// TIA Portal project "Trabajo_plantilla" (V14)
// Plantilla para la realización de la parte de programación de la asignatura de Automatización

(* hardware
DEVICE "S71500/ET200MP station_16"  S7-1500 station
   slot 0: "Perfil soporte_0"  Rack  6ES7 590-1***0-0AA0
   slot 1: "AUTO_CELDA_DE_CORTE"  CPU 1516F-3 PN/DP  6ES7 516-3FN00-0AB0  V1.8
      slot 3: "Display de la CPU_1"  6ES7591-1BA00-0AA0
   slot 2: "DI 32x24VDC BA_1"  DI 32x24VDC BA  6ES7 521-1BL10-0AA0  V1.0
   slot 3: "DQ 32x24VDC/0.5A BA_1"  DQ 32x24VDC/0.5A BA  6ES7 522-1BL10-0AA0  V1.0
   slot 4: "DI 32x24VDC BA_2"  DI 32x24VDC BA  6ES7 521-1BL10-0AA0  V1.0
*)

// ===== PLC "AUTO_CELDA_DE_CORTE"  CPU 1516F-3 PN/DP =====

VAR_GLOBAL   // PLC tag table "Tests Unitarios"
   "Tag_1" AT %M20.0 : Bool;
   "Tag_2" AT %M20.1 : Bool;
   "Tag_3" AT %M20.2 : Bool;
   "Tag_4" AT %M20.3 : Bool;
   "Tag_6" AT %M20.5 : Bool;
   "Tag_7" AT %M20.6 : Bool;
   "Tag_5" AT %M20.4 : Bool;
   "Tag_8" AT %M20.7 : Bool;
   "Tag_9" AT %M21.0 : Bool;
   "Tag_10" AT %M21.1 : Bool;
   "Tag_12" AT %MD22 : Real;
   "Tag_11" AT %M21.2 : Bool;
   "Tag_13" AT %M21.3 : Bool;
   "Tag_14" AT %M21.4 : Bool;
   "Tag_15" AT %M21.5 : Bool;
   "Tag_16" AT %M21.6 : Bool;
   "Tag_17" AT %M21.7 : Bool;
END_VAR

VAR_GLOBAL   // PLC tag table "Entradas"
   "SB2_inferior" AT %E3.5 : Bool;   // Sensor de presencia que detecta la legada de piezas al brazo 2 (derecha) desde la cinta inferior
   "SB2_superior" AT %E3.4 : Bool;   // Sensor de presencia que detecta la legada de piezas al brazo 2 (derecha) desde la cinta superior
   "SB1_inferior" AT %E3.3 : Bool;   // Sensor de presencia que detecta la legada de piezas al brazo 1 (izquierda) desde la cinta inferior
   "SB1_superior" AT %E3.2 : Bool;   // Sensor de presencia que detecta la legada de piezas al brazo 1 (izquierda) desde la cinta superior
   "pieza_válida_serigrafía" AT %E2.7 : Bool;   // Aviso del lector de códigos correspondiente de que la pieza detectada debe ser incorporada a la máquina de serigrafía
   "pieza_válida_laminado" AT %E4.1 : Bool;   // Aviso del lector de códigos correspondiente de que la pieza detectada debe ser incorporada a la máquina de laminado
   "pieza_válida_corte" AT %E4.0 : Bool;   // Aviso del lector de códigos correspondiente de que la pieza detectada debe ser incorporada a la máquina de corte
   "FC3_E" AT %E0.7 : Bool;   // Fin de carrera del pistón de alimentación de la máquina de serigrafía (expandido)
   "FC3_C" AT %E0.6 : Bool;   // Fin de carrera del pistón de alimentación de la máquina de serigrafía (comprimido)
   "FC2_E" AT %E0.5 : Bool;   // Fin de carrera del pistón de alimentación de la máquina de laminado (expandido)
   "FC2_C" AT %E0.4 : Bool;   // Fin de carrera del pistón de alimentación de la máquina de laminado (comprimido)
   "FC1_E" AT %E0.3 : Bool;   // Fin de carrera del pistón de alimentación de la máquina de corte (expandido)
   "FC1_C" AT %E0.2 : Bool;   // Fin de carrera del pistón de alimentación de la máquina de corte (comprimido)
   "SS0" AT %E4.2 : Bool;   // Sensor de presencia de la cinta de alimentación, sobre la máquina de serigrafiado
   "SL0" AT %E3.7 : Bool;   // Sensor de presencia de la cinta de alimentación, sobre la máquina de laminado
   "SC0" AT %E3.6 : Bool;   // Sensor de presencia de la cinta de alimentación, sobre la máquina de corte
   "SS3_Derecha" AT %E2.4 : Bool;   // Sensor de incorporación a la cinta de evacuación de la serigrafiadora (derecha)
   "SL3_Derecha" AT %E3.1 : Bool;   // Sensor de incorporación a la cinta de evacuación de la laminadora (derecha)
   "SC3_Derecha" AT %E3.0 : Bool;   // Sensor de incorporación a la cinta de evacuación de la máquina de corte (a la derecha)
   "MB" AT %E2.6 : Bool;   // Señal de Activación del Modo de Marcha B
   "MA" AT %E2.5 : Bool;   // Señal de Activación del Modo de Marcha A
   "OFF" AT %E0.1 : Bool;   // Señal de parada controlada
   "SS3_Izquierda" AT %E2.3 : Bool;   // Sensor de incorporación a la cinta de evacuación de la serigrafiadora (izquierda)
   "SS2" AT %E2.2 : Bool;   // Sensor a la salida de la serigrafiadora
   "SS1" AT %E2.1 : Bool;   // Sensor de presencia a la entrada de la serigrafiadora
   "SL3_Izquierda" AT %E2.0 : Bool;   // Sensor de incorporación a la cinta de evacuación de la laminadora (izquierda)
   "SL2" AT %E1.7 : Bool;   // Sensor a la salida de la laminadora
   "SL1" AT %E1.6 : Bool;   // Sensor de presencia a la entrada de la laminadora
   "SC3_Izquierda" AT %E1.5 : Bool;   // Sensor de incorporación a la cinta de evacuación de la máquina de corte (a la izquierda)
   "SC2" AT %E1.4 : Bool;   // Sensor a la salida de la máquina de corte
   "SC1" AT %E1.3 : Bool;   // Sensor de presencia a la entrada de la máquina de corte
   "ON" AT %E0.0 : Bool;   // Puesta en marcha del sistema
   "señal_pirómetro" AT %EW6 : Int;   // Señal analógica del sensor de temperatura
   "Rearme" AT %E1.0 : Bool;   // Señal de activación del rearme
   "EMER" AT %E1.1 : Bool;   // Señal de activación del estado de emergencia
END_VAR

VAR_GLOBAL   // PLC tag table "Actuadores"
   "EXTRAER_INFERIOR_B2" AT %A0.2 : Bool;   // Actuador que engloba la operación de extracción de piezas por la cinta inferior del brazo 2
   "EXTRAER_SUPERIOR_B2" AT %A0.1 : Bool;   // Actuador que engloba la operación de extracción de piezas por la cinta superior del brazo 2
   "ALIMENTAR_B2" AT %A0.0 : Bool;   // Actuador que engloba la operación de alimentación del brazo 2
   "EXTRAER_INFERIOR_B1" AT %A0.5 : Bool;   // Actuador que engloba la operación de extracción de piezas por la cinta inferior del brazo 1
   "EXTRAER_SUPERIOR_B1" AT %A0.4 : Bool;   // Actuador que engloba la operación de extracción de piezas por la cinta superior del brazo 1
   "ALIMENTAR_B1" AT %A0.3 : Bool;   // Actuador que engloba la operación de alimentación del brazo 1
   "CINTA_VOLCADO_Corte" AT %A2.2 : Bool;   // Actuador que activa la cinta de volcado de piezas de la máquina de corte
   "COMP3" AT %A1.3 : Bool;   // Actuador que efectúa la compresión del cilindro de alimentación de la máquina de serigrafía
   "EXP3" AT %A1.2 : Bool;   // Actuador que efectúa la expansión del cilindro de alimentación de la máquina de serigrafía
   "COMP2" AT %A1.1 : Bool;   // Actuador que efectúa la compresión del cilindro de alimentación de la máquina de laminado
   "EXP2" AT %A1.0 : Bool;   // Actuador que efectúa la expansión del cilindro de alimentación de la máquina de laminado
   "COMP1" AT %A0.7 : Bool;   // Actuador que efectúa la compresión del cilindro de alimentación de la máquina de corte
   "EXP1" AT %A0.6 : Bool;   // Actuador que efectúa la expansión del cilindro de alimentación de la máquina de corte
   "MÁQUINA_SERIGRAFIADO_ON" AT %A2.4 : Bool;   // Actuador que engloba el funcionamiento de la CNC de serigrafía
   "MÁQUINA_LAMINADO_ON" AT %A2.5 : Bool;   // Actuador que engloba el funcionamiento de la CNC de laminado
   "MÁQUINA_CORTE_ON" AT %A2.6 : Bool;   // Actuador que engloba el funcionamiento de la CNC de corte
   "CINTA_VOLCADO_Laminado" AT %A2.3 : Bool;   // Actuador que activa la cinta de volcado de piezas de la máquina de laminado
   "LÁMPARA_IR" AT %A2.0 : Bool;   // Lámpara infrarroja para el precalentado de piezas en la laminadora
   "CINTA_VOLCADO_Serigrafiado" AT %A2.1 : Bool;   // Actuador que activa la cinta de volcado de piezas de la máquina de serigrafiado
   "CINTA1_H" AT %A1.4 : Bool;   // Actuador que mueve la cinta 1 (superior) en sentido horario (de izquierda a derecha)
   "CINTA1_A" AT %A1.5 : Bool;   // Actuador que mueve la cinta 1 (superior) en sentido anti-horario (de derecha a izquierda)
   "CINTA2_H" AT %A1.6 : Bool;   // Actuador que mueve la cinta 2 (inferior) en sentido horario (de izquierda a derecha)
   "CINTA2_A" AT %A1.7 : Bool;   // Actuador que mueve la cinta 2 (inferior) en sentido anti-horario (de derecha a izquierda)
END_VAR

VAR_GLOBAL   // PLC tag table "Entradas (avisos)"
   "aviso_fin_tratamiento_corte" AT %E5.2 : Bool;   // Indica que la operación de corte ha concluido con éxito
   "aviso_fin_tratamiento_laminado" AT %E5.3 : Bool;   // Indica que la operación de laminado ha concluido con éxito
   "aviso_fin_tratamiento_serigrafiado" AT %E5.4 : Bool;   // Indica que la operación de serigrafiado ha concluido con éxito
   "aviso_brazo1_en_posición" AT %E4.3 : Bool;   // Señal de aviso que indica que el brazo 1 está posicionado correctamente
   "aviso_brazo2_en_posición" AT %E4.4 : Bool;   // Señal de aviso que indica que el brazo 2 está posicionado correctamente
   "aviso_fin_de_maniobra_brazo1" AT %E4.7 : Bool;   // Aviso que indica que la maniobra del brazo 1 ha concluido con éxito
   "aviso_fin_de_maniobra_brazo2" AT %E5.1 : Bool;   // Aviso que indica que la maniobra del brazo 2 ha concluido con éxito
   "aviso_máquina_corte_en_posición" AT %E5.5 : Bool;   // Aviso que indica que la máquina de corte está posicionada correctamente
   "comando_alimentar_brazo1" AT %E4.5 : Bool;   // Señal que ordena al brazo 1 a ejecutar la maniobra de alimentar
   "comando_alimentar_brazo2" AT %E4.6 : Bool;   // Señal que ordena al brazo 2 a ejecutar la maniobra de alimentar
   "aviso_máquina_laminado_en_posición" AT %E5.6 : Bool;   // Aviso que indica que la máquina de laminado está posicionada correctamente
   "aviso_máquina_serigrafiado_en_posición" AT %E5.7 : Bool;   // Aviso que indica que la máquina de serigrafiado está posicionada correctamente
END_VAR

VAR_GLOBAL   // PLC tag table "Señales Internas y Salientes"
   "aviso_Defecto_brazo1" AT %M16.1 : Bool;   // Aviso que indica que el brazo 1 se encuentra en estado de defecto
   "aviso_Defecto_brazo2" AT %M16.2 : Bool;   // Aviso que indica que el brazo 2 se encuentra en estado de defecto
   "aviso_Defecto_cinta1" AT %M13.4 : Bool;   // Aviso de que la cinta de volcado de la máquina de corte se encuentra en estado de defecto local
   "aviso_Defecto_cinta2" AT %M13.5 : Bool;   // Aviso de que la cinta de volcado de la máquina de laminado se encuentra en estado de defecto local
   "aviso_Defecto_cinta3" AT %M13.6 : Bool;   // Aviso de que la cinta de volcado de la máquina de serigrafiado se encuentra en estado de defecto local
   "aviso_Defecto_pistón1" AT %M10.4 : Bool;   // Aviso de que el pistón de alimentación de la máquina de corte ha entrado en defecto local
   "aviso_Defecto_pistón2" AT %M10.5 : Bool;   // Aviso de que el pistón de alimentación de la máquina de laminado ha entrado en defecto local
   "aviso_Defecto_pistón3" AT %M10.6 : Bool;   // Aviso de que el pistón de alimentación de la máquina deserigrafía ha entrado en defecto local
   "aviso_Standby_brazo1" AT %M15.7 : Bool;   // Aviso que indica que el brazo 1 se encuentra en espera
   "aviso_Standby_brazo2" AT %M16.0 : Bool;   // Aviso que indica que el brazo 2 se encuentra en espera
   "aviso_Standby_cinta1" AT %M13.1 : Bool;   // Aviso de que la cinta de volcado de la máquina de corte se encuentra en espera
   "aviso_Standby_cinta2" AT %M13.2 : Bool;   // Aviso de que la cinta de volcado de la máquina de laminado se encuentra en espera
   "aviso_Standby_cinta3" AT %M13.3 : Bool;   // Aviso de que la cinta de volcado de la máquina de serigrafiado se encuentra en espera
   "aviso_Standby_pistón1" AT %M10.1 : Bool;   // Aviso de que el pistón de alimentación de la máquina de corte está en estado de espera
   "aviso_Standby_pistón2" AT %M10.2 : Bool;   // Aviso de que el pistón de alimentación de la máquina de laminado está en estado de espera
   "aviso_Standby_pistón3" AT %M10.3 : Bool;   // Aviso de que el pistón de alimentación de la máquina de serigrafía está en estado de espera
   "aviso_Defecto_máquina_corte" AT %M12.6 : Bool;   // Aviso que indica que la máquina de corte se encuentra en defecto local
   "aviso_Defecto_máquina_laminado" AT %M12.7 : Bool;   // Aviso que indica que la máquina de laminado se encuentra en defecto local
   "aviso_Defecto_máquina_serigrafía" AT %M13.0 : Bool;   // Aviso que indica que la máquina de serigrafía se encuentra en defecto local
   "aviso_Standby_máquina_corte" AT %M13.7 : Bool;   // Aviso que indica que la máquina de corte está en espera
   "aviso_Standby_máquina_laminado" AT %M14.0 : Bool;   // Aviso que indica que la máquina de laminado está en espera
   "aviso_Standby_máquina_serigrafiado" AT %M14.1 : Bool;   // Aviso que indica que la máquina de serigrafiado está en espera
   "aviso_Standby_GRAL" AT %M1.5 : Bool;   // Vale 1 cuando todos los avisos de standby del sistema valen 1
   "lectura_real_pirómetro" AT %MD4 : Real;   // Lectura del pirómetro en ºC
   "mpON" AT %M0.1 : Bool;   // marca de pulso para la señal ON
   "mfON" AT %M0.0 : Bool;   // marca de flanco para la señal ON
END_VAR

VAR_GLOBAL   // PLC tag table "Marcas de Estado"
   "XON" AT %M0.2 : Bool;   // Estado de marcha del grafcet marcha_paro
   "XOFF" AT %M0.3 : Bool;   // Estado de parada controlada del grafcet marcho_parp
   "X0" AT %M0.4 : Bool;   // Estado de reposo del grafced de producción
   "X10" AT %M0.5 : Bool;   // Estado de reposo del grafcet de modos de marcha
   "XA" AT %M0.6 : Bool;   // Estado del Modo de Marcha A del GMM
   "XB" AT %M0.7 : Bool;   // Estado del Modo de Marcha B del GMM
   "X20" AT %M8.6 : Bool;   // Estado de marcha del grafcet de emergencia
   "X21" AT %M8.7 : Bool;   // Estado de emergencia del grafcet de seguridad
   "X_MA1" AT %M10.7 : Bool;   // Etapa de activación del pistón de alimentación de la máquina de corte
   "X_MA2" AT %M11.0 : Bool;   // Etapa de activación del pistón de alimentación de la máquina de laminado
   "X_MA3" AT %M11.1 : Bool;   // Etapa de activación del pistón de alimentación de la máquina de serigrafía
   "X_ME1" AT %M11.2 : Bool;   // Etapa de activación de la cinta de volcado de piezas de la máquina de corte
   "X_ME2" AT %M11.3 : Bool;   // Etapa de activación de la cinta de volcado de piezas de la máquina de laminado
   "X_ME3" AT %M11.4 : Bool;   // Etapa de activación de la cinta de volcado de piezas de la máquina de serigrafiado
   "X_MM1" AT %M11.5 : Bool;   // Etapa de activación de la máquina de corte
   "X_MM2" AT %M11.6 : Bool;   // Etapa de activación de la máquina de laminado
   "X_MM3" AT %M11.7 : Bool;   // Etapa de activación de la máquina de serigrafía
   "X_MB1" AT %M12.0 : Bool;   // Etapa de activación del brazo de carga/descarga de la izquierda
   "X_MB2" AT %M12.1 : Bool;   // Etapa de activación del brazo de carga/descarga de la derecha
   "X_Cintas" AT %M12.2 : Bool;   // Etapa de activación de las cintas de transporte principales
   "X_Defecto_GP" AT %M1.6 : Bool;   // Estado de defecto por emergencia del grafcet de producción
   "X_Trabajo" AT %M1.4 : Bool;   // Estado de trabajo que engloba los estados de todas las máquinas (su finalidad es aligerar el código)
END_VAR

DATA_BLOCK "DATOS_PRODUCCION"   // DB1
TITLE = parametros de produccion (TODOS)
{ S7_Optimized_Access := 'TRUE' }
VERSION : 0.1
// Incluye cualquier  constante numérica necesaria para el control. Este bloque se podría descomponer en varios bloques de datos temáticos si fuera necesario.
   VAR
      tiempo_exp : Time := T#20s;   // Tiempo límite para completar la maniobra de expansión (pistón)
      tiempo_comp : Time := T#20s;   // Tiempo límite para completar la maniobra de compresión (pistón)
      tiempo_serigrafiar : Time := T#20s;   // Tiempo límite para completar la operación de serigrafiado
      tiempo_cortar : Time := T#20s;   // Tiempo límite para completar la operación de cortado
      tiempo_laminar : Time := T#20s;   // Tiempo límite para completar la operación de laminado
      tiempo_brazo : Time := T#20s;   // Tiempo límite para completar una maniobra (brazo de carga/descarga)
      tiempo_evacuación : Time := T#5s;   // Tiempo mínimo para considerar que es seguro incorporar una pieza a la cinta de evacuación
      tiempo_volcado : Time := T#10s;   // Tiempo límite para mover lapieza al borde de la cinta de volcado.
      tiempo_parada_controlada : Time := T#15s;   // Tiempo mínimo para detenerse el sistema tras la activación de la señal OFF
      temp_referencia_laminado : Real := 100.0;   // Temperatura a la que se deberá mantener la pieza durante el proceso de laminado. Si se introduce una temperatura menor a la ambiente, no se encenderá la lámpara IR.
      lim_sup_pirómetro : Real := 350.0;   // Límite superior del campo de medida del pirómetro
      lim_inf_pirómetro : Real := -20.0;   // Límite inferior del campo de medida del pirómetro
      flag_sentido_cinta_superior : Bool := False;   // Será ==TRUE cuando la cinta de alimentación (superior) se mueva de izquierda a derecha (sentido horario)
      flag_sentido_cinta_inferior : Bool := True;   // Será ==TRUE cuando la cinta de evacuaciónn (inferior) se mueva de izquierda a derecha (sentido anti-horario)
      flag_brazo1_alimentar : Bool := False;   // Será ==TRUE cuando se desee que el brazo 1 alimente la cinta superior
      flag_brazo1_extracción_superior : Bool := True;   // Será ==TRUE cuando se desee que el brazo 1 descargue piezas por la cinta superior
      flag_brazo1_extracción_inferior : Bool := False;   // Será ==TRUE cuando se desee que el brazo 1 descargue piezas por la cinta inferior
      flag_brazo2_alimentar : Bool := True;   // Será ==TRUE cuando se desee que el brazo 2 alimente la cinta superior
      flag_brazo2_extracción_superior : Bool := False;   // Será ==TRUE cuando se desee que el brazo 2 descargue piezas por la cinta superior
      flag_brazo2_extracción_inferior : Bool := True;   // Será ==TRUE cuando se desee que el brazo 2 descargue piezas por la cinta inferior
   END_VAR
BEGIN
END_DATA_BLOCK

DATA_BLOCK "DATOS_PRODUCCION_MODO_A"   // DB4
TITLE = parametros de producción MODO_A
{ S7_Optimized_Access := 'TRUE' }
VERSION : 0.1
// subconjunto de parámetros de DATOS_PRODUCCION (DB1)
   VAR
      temp_ref_laminado : Real := 150.0;   // Tamperatura a la que se desea mantener la pieza durante el laminado
      flag_sentido_cinta_superior : Bool := false;   // Será ==TRUE cuando la cinta de alimentación (superior) se mueva de izquierda a derecha (sentido horario)
      flag_sentido_cinta_inferior : Bool := true;   // Será ==TRUE cuando la cinta de evacuaciónn (inferior) se mueva de izquierda a derecha (sentido anti-horario)
      flag_brazo1_alimentar : Bool := false;   // Será ==TRUE cuando se desee que el brazo 1 alimente la cinta superior
      flag_brazo1_extracción_superior : Bool := true;   // Será ==TRUE cuando se desee que el brazo 1 descargue piezas por la cinta superior
      flag_brazo1_extracción_inferior : Bool := false;   // Será ==TRUE cuando se desee que el brazo 1 descargue piezas por la cinta inferior
      flag_brazo2_alimentar : Bool := true;   // Será ==TRUE cuando se desee que el brazo 2 alimente la cinta superior
      flag_brazo2_extracción_superior : Bool := false;   // Será ==TRUE cuando se desee que el brazo 2 descargue piezas por la cinta superior
      flag_brazo2_extracción_inferior : Bool := true;   // Será ==TRUE cuando se desee que el brazo 2 descargue piezas por la cinta inferior
   END_VAR
BEGIN
END_DATA_BLOCK

DATA_BLOCK "DATOS_PRODUCCION_MODO_B"   // DB5
TITLE = parámetros de producción modo B
{ S7_Optimized_Access := 'TRUE' }
VERSION : 0.1
// subconjunto de todos los parámetros de producción (DB1)
   VAR
      temp_ref_laminado : Real := 250.0;   // Tamperatura a la que se desea mantener la pieza durante el laminado
      flag_sentido_cinta_superior : Bool := true;   // Será ==TRUE cuando la cinta de alimentación (superior) se mueva de izquierda a derecha (sentido horario)
      flag_sentido_cinta_inferior : Bool := false;   // Será ==TRUE cuando la cinta de evacuaciónn (inferior) se mueva de izquierda a derecha (sentido anti-horario)
      flag_brazo1_alimentar : Bool := true;   // Será ==TRUE cuando se desee que el brazo 1 alimente la cinta superior
      flag_brazo1_extracción_superior : Bool := false;   // Será ==TRUE cuando se desee que el brazo 1 descargue piezas por la cinta superior
      flag_brazo1_extracción_inferior : Bool := true;   // Será ==TRUE cuando se desee que el brazo 1 descargue piezas por la cinta inferior
      flag_brazo2_alimentar : Bool := false;   // Será ==TRUE cuando se desee que el brazo 2 alimente la cinta superior
      flag_brazo2_extracción_superior : Bool := true;   // Será ==TRUE cuando se desee que el brazo 2 descargue piezas por la cinta superior
      flag_brazo2_extracción_inferior : Bool := false;   // Será ==TRUE cuando se desee que el brazo 2 descargue piezas por la cinta inferior
   END_VAR
BEGIN
END_DATA_BLOCK

// folder: Máquinas/Bloques de Datos

DATA_BLOCK "Sistema de Alimentación_DB"   // DB12
{ S7_Optimized_Access := 'TRUE' }
VERSION : 0.1
// stored: InstanceOfName Sistema de Alimentación
"Sistema de Alimentación"
BEGIN
END_DATA_BLOCK

DATA_BLOCK "Sistema de Volcado_DB"   // DB13
{ S7_Optimized_Access := 'TRUE' }
VERSION : 0.1
// stored: InstanceOfName Sistema de Volcado
"Sistema de Volcado"
BEGIN
END_DATA_BLOCK

DATA_BLOCK "Brazo1_(Izquierdo)_DB"   // DB14
{ S7_Optimized_Access := 'TRUE' }
VERSION : 0.1
// stored: InstanceOfName Brazo de Carga/Descarga
"Brazo de Carga/Descarga"
BEGIN
END_DATA_BLOCK

DATA_BLOCK "Brazo2_(Derecho)_DB"   // DB15
{ S7_Optimized_Access := 'TRUE' }
VERSION : 0.1
// stored: InstanceOfName Brazo de Carga/Descarga
"Brazo de Carga/Descarga"
BEGIN
END_DATA_BLOCK

DATA_BLOCK "CNC (Corte)_DB"   // DB16
{ S7_Optimized_Access := 'TRUE' }
VERSION : 0.1
// stored: InstanceOfName CNC (Corte/Serigrafía)
"CNC (Corte/Serigrafía)"
BEGIN
END_DATA_BLOCK

DATA_BLOCK "CNC (Laminado)_DB"   // DB17
{ S7_Optimized_Access := 'TRUE' }
VERSION : 0.1
// stored: InstanceOfName CNC (Laminado)
"CNC (Laminado)"
BEGIN
END_DATA_BLOCK

DATA_BLOCK "CNC (Serigrafía)_DB"   // DB18
{ S7_Optimized_Access := 'TRUE' }
VERSION : 0.1
// stored: InstanceOfName CNC (Corte/Serigrafía)
"CNC (Corte/Serigrafía)"
BEGIN
END_DATA_BLOCK

// folder: System blocks/Program resources

DATA_BLOCK "TON_PARADA_Controlada_DB"   // DB19
{ S7_Optimized_Access := 'TRUE' }
AUTHOR : Simatic
FAMILY : IEC
NAME : IEC_TMR
VERSION : 1.0
// stored: InstanceOfName IEC_TIMER
"IEC_TIMER"
BEGIN
END_DATA_BLOCK

// folder: Tests

DATA_BLOCK "Pistón (Máquina)_test_DB"   // DB2
{ S7_Optimized_Access := 'TRUE' }
VERSION : 0.1
// stored: InstanceOfName Pistón (Máquina)
"Pistón (Máquina)"
BEGIN
END_DATA_BLOCK

DATA_BLOCK "Pistón (Maniobra Simple)_test_DB"   // DB3
{ S7_Optimized_Access := 'TRUE' }
VERSION : 0.1
// stored: InstanceOfName Pistón (Maniobra Simple)
"Pistón (Maniobra Simple)"
BEGIN
END_DATA_BLOCK

DATA_BLOCK "CNC_Corte_test_DB"   // DB6
{ S7_Optimized_Access := 'TRUE' }
VERSION : 0.1
// stored: InstanceOfName CNC (Corte/Serigrafía)
"CNC (Corte/Serigrafía)"
BEGIN
END_DATA_BLOCK

DATA_BLOCK "CNC (Laminado)_test_DB"   // DB7
{ S7_Optimized_Access := 'TRUE' }
VERSION : 0.1
// stored: InstanceOfName CNC (Laminado)
"CNC (Laminado)"
BEGIN
END_DATA_BLOCK

DATA_BLOCK "Brazo de Carga/Descarga_test_DB"   // DB8
{ S7_Optimized_Access := 'TRUE' }
VERSION : 0.1
// stored: InstanceOfName Brazo de Carga/Descarga
"Brazo de Carga/Descarga"
BEGIN
END_DATA_BLOCK

DATA_BLOCK "Cinta de Volcado (Aviso de Disponibilidad)_test_DB"   // DB9
{ S7_Optimized_Access := 'TRUE' }
VERSION : 0.1
// stored: InstanceOfName Cinta de Volcado (Aviso de Disponibilidad)
"Cinta de Volcado (Aviso de Disponibilidad)"
BEGIN
END_DATA_BLOCK

DATA_BLOCK "Cinta de Volcado (Máquina)_test_DB"   // DB10
{ S7_Optimized_Access := 'TRUE' }
VERSION : 0.1
// stored: InstanceOfName Cinta de Volcado (Máquina)
"Cinta de Volcado (Máquina)"
BEGIN
END_DATA_BLOCK

// folder: (top level)

ORGANIZATION_BLOCK "Main"   // OB1, LAD, ProgramCycle
TITLE = "Main Program Sweep (Cycle)"
{ S7_Optimized_Access := 'TRUE' }
VERSION : 0.1
// Contenido del  Programa Principal:
// A)  Segmentos con llamadas incondicionales a otros bloques por orden de prioridad (GEMER, MODOS DE MARCHA, FLANCOS y CONECTORES, ANALOGICA ,  bloques TIPO MÁQUINA) .
// 
// B) Grafcet de Producción "GP"
   VAR_INPUT
      Initial_Call : Bool;   // Initial call of this OB
      Remanence : Bool;   // =True, if remanent data are available
   END_VAR
   VAR_TEMP
      error_lectura_pirómetro : Bool;   // Aviso de error de lectura del pirómetro
   END_VAR
BEGIN

REGION Network 1 (STL): Tests Unitarios
   // CALL  "test_unitario_maquina_pistón"
   // CALL  "test_unitario_maniobra_pistón"
   // CALL  "test_unitario_máquina_laminado"
   // CALL  "test_unitario_máquina_brazo"
   // CALL  "test_unitario_disponibilidad_cinta_de_evacuación"
   // CALL  "test_unitario_máquina_cinta_de_volcado"
   // CALL  "test_unitario_máquina_corte"
END_REGION

REGION Network 2 (STL): LLamada a Bloques de Metacontrol
         CALL  "grafcet_marcha_y_parada_controlada_(GMPC)";
         CALL  "grafcet_modos_de_marcha_(GMM)";
         CALL  "grafcet_seguridad_(GEMER)";
END_REGION

REGION Network 3 (STL): Llamada a Bloques de Manejo de Señales
         CALL  "flancos_y_conectores";
         CALL  "tratamiento_señal_pirómetro"
         ( RAW                := "señal_pirómetro",
           BIPOLAR            := FALSE,
           HI_LIM             := "DATOS_PRODUCCION".lim_sup_pirómetro,
           LO_LIM             := "DATOS_PRODUCCION".lim_inf_pirómetro,
           RESET              := FALSE,
           lectura_valor_real := "lectura_real_pirómetro",
           error              := #error_lectura_pirómetro
         );
END_REGION

REGION Network 4 (STL): Llamada a las Máquinas
         CALL  "Sistema de Alimentación", "Sistema de Alimentación_DB";
         CALL  "Sistema de Volcado", "Sistema de Volcado_DB";
         CALL  "Brazo de Carga/Descarga", "Brazo1_(Izquierdo)_DB"
         ( Start              := "X_MB1",
           EMER               := "X21",
           tiempo             := "DATOS_PRODUCCION".tiempo_brazo,
           brazo_en_posición  := "aviso_brazo1_en_posición",
           Rearme             := "X20",
           S_superior         := "SB1_superior",
           S_inferior         := "SB1_inferior",
           fin_maniobra       := "aviso_fin_de_maniobra_brazo1",
           orden_alimentar    := "comando_alimentar_brazo1",
           flag_alim          := "DATOS_PRODUCCION".flag_brazo1_alimentar,
           flag_extr_inf      := "DATOS_PRODUCCION".flag_brazo1_extracción_inferior,
           flag_extr_sup      := "DATOS_PRODUCCION".flag_brazo1_extracción_superior,
           aviso_standby      := "aviso_Standby_brazo1",
           ALIMENTAR          := "ALIMENTAR_B1",
           EXTRAER_POR_ARRIBA := "EXTRAER_SUPERIOR_B1",
           EXTRAER_POR_DEBAJO := "EXTRAER_INFERIOR_B1",
           aviso_defecto      := "aviso_Defecto_brazo1"
         );
         CALL  "Brazo de Carga/Descarga", "Brazo2_(Derecho)_DB"
         ( Start              := "X_MB2",
           EMER               := "X21",
           tiempo             := "DATOS_PRODUCCION".tiempo_brazo,
           brazo_en_posición  := "aviso_brazo2_en_posición",
           Rearme             := "X20",
           S_superior         := "SB2_superior",
           S_inferior         := "SB2_inferior",
           fin_maniobra       := "aviso_fin_de_maniobra_brazo2",
           orden_alimentar    := "comando_alimentar_brazo2",
           flag_alim          := "DATOS_PRODUCCION".flag_brazo2_alimentar,
           flag_extr_inf      := "DATOS_PRODUCCION".flag_brazo2_extracción_inferior,
           flag_extr_sup      := "DATOS_PRODUCCION".flag_brazo2_extracción_superior,
           aviso_standby      := "aviso_Standby_brazo2",
           ALIMENTAR          := "ALIMENTAR_B2",
           EXTRAER_POR_ARRIBA := "EXTRAER_SUPERIOR_B2",
           EXTRAER_POR_DEBAJO := "EXTRAER_INFERIOR_B2",
           aviso_defecto      := "aviso_Defecto_brazo2"
         );
         CALL  "CNC (Corte/Serigrafía)", "CNC (Corte)_DB"
         ( Start               := "X_MM1",
           EMER                := "X21",
           SE                  := "SC1",
           máquina_en_posición := "aviso_máquina_corte_en_posición",
           Rearme              := "X20",
           tiempo_límite       := "DATOS_PRODUCCION".tiempo_cortar,
           MÁQUINA_ON          := "MÁQUINA_CORTE_ON",
           aviso_standby       := "aviso_Standby_máquina_corte",
           aviso_defecto       := "aviso_Defecto_máquina_corte"
         );
         CALL  "CNC (Laminado)", "CNC (Laminado)_DB"
         ( Start               := "X_MM2",
           EMER                := "X21",
           tiempo              := "DATOS_PRODUCCION".tiempo_laminar,
           máquina_en_posición := "aviso_máquina_laminado_en_posición",
           Rearme              := "X20",
           error_lectura_piro  := #error_lectura_pirómetro,
           SE                  := "SL1",
           lectura_pirómetro   := "lectura_real_pirómetro",
           T_ref               := "DATOS_PRODUCCION".temp_referencia_laminado,
           aviso_standby       := "aviso_Standby_máquina_laminado",
           MÁQUINA_ON          := "MÁQUINA_LAMINADO_ON",
           LÁMPARA_IR_ON       := "LÁMPARA_IR",
           aviso_defecto       := "aviso_Defecto_máquina_laminado"
         );
         CALL  "CNC (Corte/Serigrafía)", "CNC (Serigrafía)_DB"
         ( Start               := "X_MM3",
           EMER                := "X21",
           SE                  := "SS1",
           máquina_en_posición := "aviso_máquina_serigrafiado_en_posición",
           Rearme              := "X20",
           tiempo_límite       := "DATOS_PRODUCCION".tiempo_serigrafiar,
           MÁQUINA_ON          := "MÁQUINA_SERIGRAFIADO_ON",
           aviso_standby       := "aviso_Standby_máquina_serigrafiado",
           aviso_defecto       := "aviso_Defecto_máquina_serigrafía"
         );
END_REGION

REGION Network 5 (STL): Simplificación "X_Trabajo "
   // Para aligerar el código se ha creado esta marcha de estado que representa el paralelo de todas las máquinas.
         A     "X_Trabajo";
         =     "X_MA1";
         =     "X_MA2";
         =     "X_MA3";
         =     "X_MB1";
         =     "X_MB2";
         =     "X_ME1";
         =     "X_ME2";
         =     "X_ME3";
         =     "X_MM1";
         =     "X_MM2";
         =     "X_MM3";
         =     "X_Cintas";
END_REGION

REGION Network 6 (STL): Simplificación Avisos de Standby
         A     "aviso_Standby_brazo1";
         A     "aviso_Standby_brazo2";
         A     "aviso_Standby_cinta1";
         A     "aviso_Standby_cinta2";
         A     "aviso_Standby_cinta3";
         A     "aviso_Standby_máquina_corte";
         A     "aviso_Standby_máquina_laminado";
         A     "aviso_Standby_máquina_serigrafiado";
         A     "aviso_Standby_pistón1";
         A     "aviso_Standby_pistón2";
         A     "aviso_Standby_pistón3";
         =     "aviso_Standby_GRAL";
END_REGION

REGION Network 7 (STL): X0->Trabajo (Arranque)
   // Acceso a todas las etapas de trabajo de las máquinas
         A     "X0";
         A     "XON";
         R     "X0";
         S     "X_Trabajo";
END_REGION

REGION Network 8 (STL): X_Trabajo->X0 (Parada Controlada)
   // Cuando transcurre el tiempo mínimo asignado y todas las máquinas están en standby, se vuelve al estado de reposo del sistema.
         A     "X_Trabajo";
         A     "TON_PARADA_Controlada_DB".Q;
         A     "aviso_Standby_GRAL";
         R     "X_Trabajo";
         S     "X0";
END_REGION

REGION Network 9: Gestión Cintas de Transporte Principales
   // Según el modo de marcha, las cintas se moverán en un sentido o en otro.
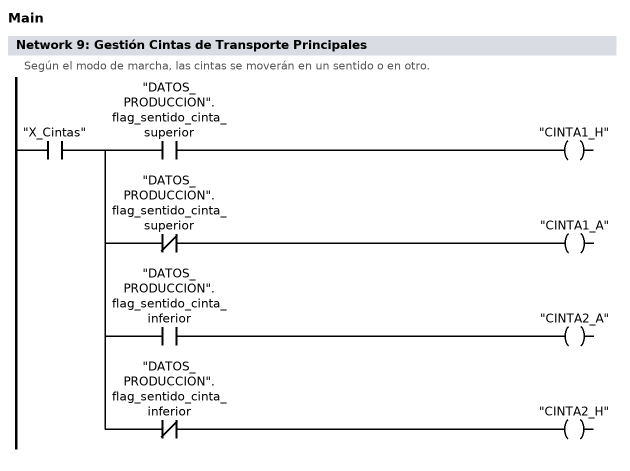
   RUNG wire#powerrail
      Contact( "X_Cintas" )
      wire#w1
      Contact( "DATOS_PRODUCCION".flag_sentido_cinta_superior )
      Coil( "CINTA1_H" )
   END_RUNG
   RUNG wire#w1
      I_Contact( "DATOS_PRODUCCION".flag_sentido_cinta_superior )
      Coil( "CINTA1_A" )
   END_RUNG
   RUNG wire#w1
      Contact( "DATOS_PRODUCCION".flag_sentido_cinta_inferior )
      Coil( "CINTA2_A" )
   END_RUNG
   RUNG wire#w1
      I_Contact( "DATOS_PRODUCCION".flag_sentido_cinta_inferior )
      Coil( "CINTA2_H" )
   END_RUNG
   // the same network as SCL:
   "CINTA1_H" := "X_Cintas" AND "DATOS_PRODUCCION".flag_sentido_cinta_superior;
   "CINTA1_A" := "X_Cintas" AND NOT "DATOS_PRODUCCION".flag_sentido_cinta_superior;
   "CINTA2_A" := "X_Cintas" AND "DATOS_PRODUCCION".flag_sentido_cinta_inferior;
   "CINTA2_H" := "X_Cintas" AND NOT "DATOS_PRODUCCION".flag_sentido_cinta_inferior;
END_REGION
END_ORGANIZATION_BLOCK

ORGANIZATION_BLOCK "Startup"   // OB100, LAD, Startup
TITLE = "Complete Restart"
{ S7_Optimized_Access := 'TRUE' }
VERSION : 0.1
// Bloque de arranque: se ejecuta una única vez antes del bloque OB1
   VAR_INPUT
      LostRetentive : Bool;   // True if retentive data are lost
      LostRTC : Bool;   // True if date and time are lost
   END_VAR
BEGIN

REGION Network 1 (STL): ARRANQUE
         SET;
         R     "XON";
         R     "X21";
         R     "XA";
         R     "XB";
         R     "X_Cintas";
         R     "X_Trabajo";
         R     "X_Defecto_GP";
         R     "X_MA1";
         R     "X_MA2";
         R     "X_MA3";
         R     "X_MB1";
         R     "X_MB2";
         R     "X_ME1";
         R     "X_ME2";
         R     "X_ME3";
         R     "X_MM1";
         R     "X_MM2";
         R     "X_MM3";
         S     "X0";
         S     "X10";
         S     "X20";
         S     "XOFF";
END_REGION
END_ORGANIZATION_BLOCK

// folder: Analógico

FUNCTION "tratamiento_señal_pirómetro" : Void   // FC8, LAD
TITLE = Tratamiento de sensor analógico con entrada RESET
{ S7_Optimized_Access := 'TRUE' }
VERSION : 0.1
// 1. Aviso de error cuando el valor de entrada (RAW) está en los valores máximos o mínimos de campo de trabajo del sensor.
// 2. Emplea SCALE (FC_105) para la conversión a  ºC  de la entrada (RAW)
// 3. RESET funciona por nivel. Mienstras RESET:=TRUE todas las salidas quedan a nivel bajo.
// 4. El transductir hace medidas en el rango de -20 ºC a 350 ºC.
// 5. La señal en bruto está comprendida entre 0 y 27648.
   VAR_INPUT
      RAW : Int;   // señal transducida según llega de la periferia
      BIPOLAR : Bool;   // TRUE +- 27.648 valores, FALSE +27.648 valores
      HI_LIM : Real;   // valor máximo del campo de trabajo del sensor
      LO_LIM : Real;   // valor mínimo del campo de trabajo del sensor
      RESET : Bool;   // todas las salidas a nivel bajo
   END_VAR
   VAR_OUTPUT
      lectura_valor_real : Real;
      error : Bool;   // valor medido en máximos o mínimos del campo de trabajo
   END_VAR
   VAR_TEMP
      retSCALE : Word;   // valor de retorno de la función SCALE (FC-105)
   END_VAR
BEGIN

REGION Network 1 (STL): RESET
   // Funciona por nivel. Mientras esté activo el bloque no proporciona salidas válidas
         A     #RESET;
         R     #error;
         JCN   _RES;
         L     0.0;
         T     #lectura_valor_real;
   _RES: NOP   0;
         A     #RESET;
         BEC;
END_REGION

REGION Network 2: LLamada a bloque SCALE
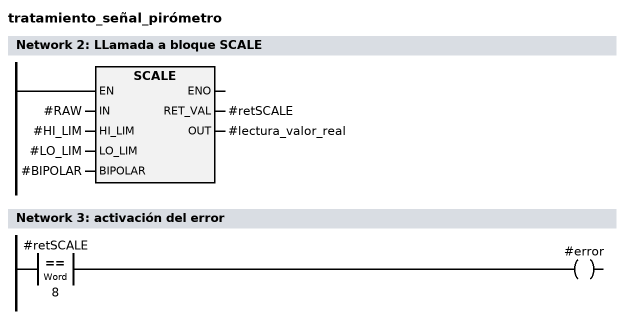
   #retSCALE := SCALE(IN := #RAW,
                      HI_LIM := #HI_LIM,
                      LO_LIM := #LO_LIM,
                      BIPOLAR := #BIPOLAR,
                      OUT => #lectura_valor_real);
END_REGION

REGION Network 3: activación del error
   RUNG wire#powerrail
      { S7_Templates := "SrcType := Word" } EQ_Contact(in1 := #retSCALE, in2 := 8)
      Coil( #error )
   END_RUNG
   // the same network as SCL:
   #error := #retSCALE = 8;
END_REGION
END_FUNCTION

// folder: Flancos

FUNCTION "flancos_y_conectores" : Void   // FC3, LAD
TITLE = gestión de flancos y conectores
{ S7_Optimized_Access := 'TRUE' }
VERSION : 0.1
// Flancos: un segmento por cada señal digital para determinar una marca de pulso (ejemplos:  evaluar si se ha producido un flanco positivo del interruptor de marcha, de un detector óptico etc. )
// 
// Conectores: un segmento por cada marca auxiliar global que hay que evaluar (por ejemplo: detector auxiliar de que una pieza ha pasado por varias celdas etc.)
BEGIN

REGION Network 1: ejemplo: flanco de subida señal de puesta en marcha- ON
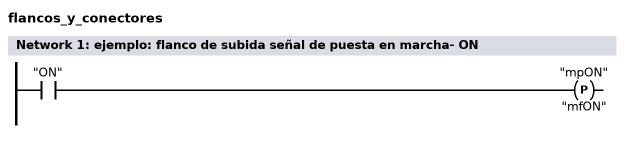
   "mpON" := "ON" AND NOT "mfON";   // rising edge
   "mfON" := "ON";
END_REGION
END_FUNCTION

// folder: Maniobras

FUNCTION_BLOCK "Pistón (Maniobra Simple)"   // FB3, LAD
TITLE = Maniobra simple con gestión de error por tiempo límite
{ S7_Optimized_Access := 'TRUE' }
VERSION : 0.1
// Se asume que la condición de inicio es TRUE. Será responsabilidad del usuario llamar a la maniobra sólo cuando se haya cumplido dicha condición. Tras la DESCONEXIÓN, el bloque queda listo para volver a ser llamado, no es necesario reiniciarlo.
// (BLOQUE AUTOCONTENIDO)
   VAR_INPUT
      SFIN : Bool;   // detector de finalización de maniobra
      tiempo_limite : Time;   // tiempo máximo de duración
      RESET : Bool;   // entrada asíncrona, parada brusca de maniobra
   END_VAR
   VAR_OUTPUT
      ACT : Bool;   // actuador de maniobra
      aviso_error_tiempo_limite : Bool;
      aviso_fin_maniobra : Bool;
   END_VAR
   VAR
      X_MAN : Bool;   // estado_maniobra_activa
      X_error_tiempo_limite : Bool;
      X_fin_maniobra : Bool;
      bit_de_trabajo : Bool;   // plantilla arranque
      temporizador : TON_TIME;
   END_VAR
BEGIN

REGION Network 1 (STL): DESCONEXION RESET (prioridad máxima)
   // Desconexión prioritaria.
         A     #RESET;
         JCN   _007;
         CALL  RESET_TIMER
         ( "TIMER" := #temporizador
         );
         A     #RESET;
         R     #bit_de_trabajo;
         R     #aviso_error_tiempo_limite;
         R     #aviso_fin_maniobra;
         R     #ACT;
         BEC;
   _007: NOP   0;
END_REGION

REGION Network 2 (STL): DESCONEXIÓN error tiempo limite
   // Desconexión Prioritaria. Se deja el bloque listo para ser llamado en el futuro.
         A     #X_error_tiempo_limite;
         JCN   _005;
         CALL  RESET_TIMER
         ( "TIMER" := #temporizador
         );
         A     #X_error_tiempo_limite;
         R     #bit_de_trabajo;
         R     #ACT;
         R     #aviso_fin_maniobra;
         R     #X_error_tiempo_limite;
         S     #aviso_error_tiempo_limite;
         BEC;
   _005: NOP   0;
END_REGION

REGION Network 3 (STL): DESCONEXIÓN fin de maniobra
   // Desconexión Prioritaria. Se deja el bloque listo para ser llamado en el futuro.
         A     #X_fin_maniobra;
         JCN   _006;
         CALL  RESET_TIMER
         ( "TIMER" := #temporizador
         );
         A     #X_fin_maniobra;
         R     #bit_de_trabajo;
         R     #ACT;
         R     #aviso_error_tiempo_limite;
         R     #X_fin_maniobra;
         S     #aviso_fin_maniobra;
         BEC;
   _006: NOP   0;
END_REGION

REGION Network 4 (STL): CONEXIÓN: activación de X_MAN (maniobra simple)
   // Arrancamos la maniobra y eliminamos los avisos externos. Se trata de un arranque directo con la llamada a la maniobra, sin comprobación de condiciones de arranque. Será responsabilidad del usuario llamar a la maniobra cuando se hayan cumplido las condiciones de inicio necesarias.
         SET;
         FP    #bit_de_trabajo;
         S     #X_MAN;
         R     #aviso_error_tiempo_limite;
         R     #aviso_fin_maniobra;
         R     #X_error_tiempo_limite;
         R     #X_fin_maniobra;
END_REGION

REGION Network 5 (STL): CONFIGURACIÓN TEMPORIZADOR
   // Emplearemos un temporizador IEC TON.
         CALL  #temporizador
         ( IN := #X_MAN,
           PT := #tiempo_limite,
           Q  := ,
           ET :=
         );
END_REGION

REGION Network 6 (STL): activación aviso interno error de tiempo
         A     #X_MAN;
         A     #temporizador.Q;
         S     #X_error_tiempo_limite;
         R     #X_MAN;
END_REGION

REGION Network 7: activación aviso interno fin de maniobra
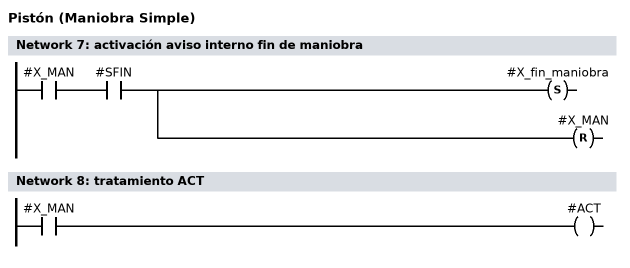
   RUNG wire#powerrail
      Contact( #X_MAN )
      Contact( #SFIN )
      wire#w1
      S_Coil( #X_fin_maniobra )
   END_RUNG
   RUNG wire#w1
      R_Coil( #X_MAN )
   END_RUNG
   // the same network as SCL:
   IF #X_MAN AND #SFIN THEN
       #X_fin_maniobra := TRUE;
       #X_MAN := FALSE;
   END_IF;
END_REGION

REGION Network 8: tratamiento ACT
   RUNG wire#powerrail
      Contact( #X_MAN )
      Coil( #ACT )
   END_RUNG
   // the same network as SCL:
   #ACT := #X_MAN;
END_REGION
END_FUNCTION_BLOCK

// folder: Metacontrol

FUNCTION "grafcet_seguridad_(GEMER)" : Void   // FC4, LAD
TITLE = grafcet para la gestión de parada brusca- paso a defecto seta EMER
{ S7_Optimized_Access := 'TRUE' }
VERSION : 0.1
// Se fuerza el GP a un estado de defecto global, y a los grafcets GMPC y GMM a sus correspondientes estados de reposo (apagado). Para implementar el forzado y evitar conflictos con los arranques de los grafcets GMPC y GMM, se ha incluido en las transiciones de arranque de los mismos como condición "X21" negada. Cuando se desenclave "X21", dichos grafcets podrán arrancar con normalidad.
// Para gestionar la emergencia y rearme de las máquinas se ha empleado como señal de emergencia y rearme las marcas "X21" y "X20" en la llamada incondicional a cada máquina que se realiza en el segmento 4 del MAIN. Internamente, cada máquina avisa de la emergencia a sus maniobras.
BEGIN

REGION Network 1 (STL): X20->X21 (Activación EMER)
         A     "X20";
         A     "EMER";
         R     "X20";
         S     "X21";
END_REGION

REGION Network 2 (STL): X21->X20 (Rearme)
         A     "X21";
         AN    "EMER";
         A     "Rearme";
         R     "X21";
         S     "X20";
END_REGION

REGION Network 3 (STL): Tratamiento del defecto - Forzado GP
   // Accede al estado de defecto
         A     "X21";
         R     "X0";
         R     "X_Trabajo";
         S     "X_Defecto_GP";
END_REGION

REGION Network 4 (STL): Tratamiento del defecto - Forzado GMM
   // Se fuerza el estado de reposo del GMM. Se ha incluido en las transiciones de arranque del GMM la marca X21 negada para que no haya conflicto.
         A     "X21";
         R     "XA";
         R     "XB";
         S     "X10";
END_REGION

REGION Network 5 (STL): Tratamiento del defecto - Forzado GMPC
   // En el arranque del GMPC se ha incluido como condición la marca "X21" negada para que no haya conflicto con el forzado.
         A     "X21";
         R     "XON";
         S     "XOFF";
END_REGION

REGION Network 6 (STL): Tratamiento Rearme.
   // Se informa a las máquinas del rearme a través del segmento 4 del MAIN (como señal de emergencia se ha usado la marca "X21", y como señal de rearme la marca "X20".
         A     "X_Defecto_GP";
         A     "X20";
         R     "X_Defecto_GP";
         S     "X0";
END_REGION
END_FUNCTION

FUNCTION "grafcet_modos_de_marcha_(GMM)" : Void   // FC5, LAD
TITLE = Grafcet que gestiona 2 modos de marcha: A y B
{ S7_Optimized_Access := 'TRUE' }
VERSION : 0.1
// Según los bloques DB que se incluyen:
// -Modo A: La cinta superior se mueve hacia la izquierda y la inferior hacia la derecha, de modo que el brazo 2 alimenta piezas por arriba y las retira por debajo, y el brazo 1 las retira por arriba. La temperatura de laminado es de 150ºC. 
// -Modo B: La cinta superior se mueve hacia la derecha y la inferior hacia la izquierda, de modo que el brazo 1 alimenta por arriba y descarga por debajo, y el brazo 2 sólo descarga por arriba. La temperatura de laminado es de 250ºC.
// 
// NOTA: aunque no se ha restringido la opción, no se recomienta cambiar el modo de marcha mietras el sistema esté en funcionamiento, ya que al afectar al sentido de las cintas podrían provocarse colisiones en la cinta de evacuación.
BEGIN

REGION Network 1: Tratamiento Modo de Marcha A
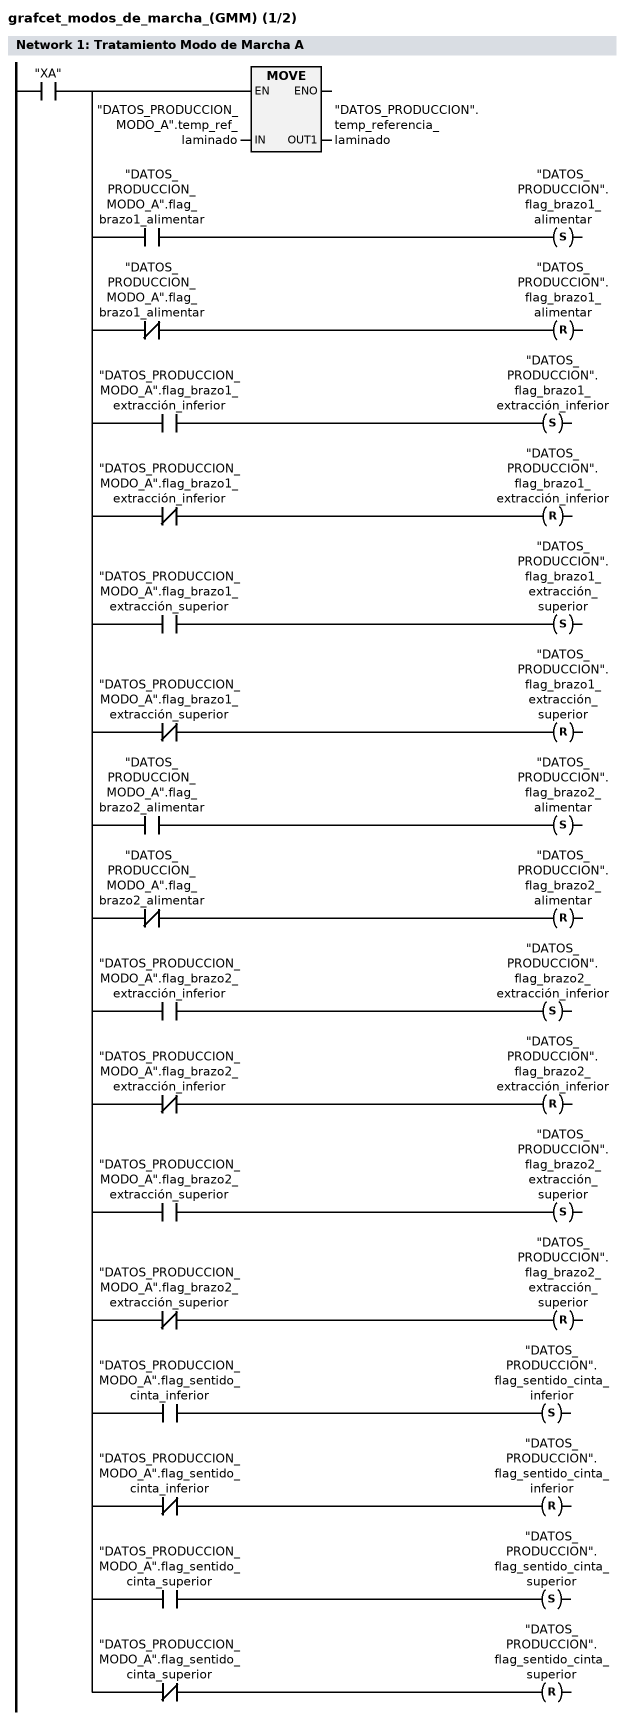
   RUNG wire#powerrail
      Contact( "XA" )
      wire#w1
      Move(in := "DATOS_PRODUCCION_MODO_A".temp_ref_laminado, out1 => "DATOS_PRODUCCION".temp_referencia_laminado)
   END_RUNG
   RUNG wire#w1
      Contact( "DATOS_PRODUCCION_MODO_A".flag_brazo1_alimentar )
      S_Coil( "DATOS_PRODUCCION".flag_brazo1_alimentar )
   END_RUNG
   RUNG wire#w1
      I_Contact( "DATOS_PRODUCCION_MODO_A".flag_brazo1_alimentar )
      R_Coil( "DATOS_PRODUCCION".flag_brazo1_alimentar )
   END_RUNG
   RUNG wire#w1
      Contact( "DATOS_PRODUCCION_MODO_A".flag_brazo1_extracción_inferior )
      S_Coil( "DATOS_PRODUCCION".flag_brazo1_extracción_inferior )
   END_RUNG
   RUNG wire#w1
      I_Contact( "DATOS_PRODUCCION_MODO_A".flag_brazo1_extracción_inferior )
      R_Coil( "DATOS_PRODUCCION".flag_brazo1_extracción_inferior )
   END_RUNG
   RUNG wire#w1
      Contact( "DATOS_PRODUCCION_MODO_A".flag_brazo1_extracción_superior )
      S_Coil( "DATOS_PRODUCCION".flag_brazo1_extracción_superior )
   END_RUNG
   RUNG wire#w1
      I_Contact( "DATOS_PRODUCCION_MODO_A".flag_brazo1_extracción_superior )
      R_Coil( "DATOS_PRODUCCION".flag_brazo1_extracción_superior )
   END_RUNG
   RUNG wire#w1
      Contact( "DATOS_PRODUCCION_MODO_A".flag_brazo2_alimentar )
      S_Coil( "DATOS_PRODUCCION".flag_brazo2_alimentar )
   END_RUNG
   RUNG wire#w1
      I_Contact( "DATOS_PRODUCCION_MODO_A".flag_brazo2_alimentar )
      R_Coil( "DATOS_PRODUCCION".flag_brazo2_alimentar )
   END_RUNG
   RUNG wire#w1
      Contact( "DATOS_PRODUCCION_MODO_A".flag_brazo2_extracción_inferior )
      S_Coil( "DATOS_PRODUCCION".flag_brazo2_extracción_inferior )
   END_RUNG
   RUNG wire#w1
      I_Contact( "DATOS_PRODUCCION_MODO_A".flag_brazo2_extracción_inferior )
      R_Coil( "DATOS_PRODUCCION".flag_brazo2_extracción_inferior )
   END_RUNG
   RUNG wire#w1
      Contact( "DATOS_PRODUCCION_MODO_A".flag_brazo2_extracción_superior )
      S_Coil( "DATOS_PRODUCCION".flag_brazo2_extracción_superior )
   END_RUNG
   RUNG wire#w1
      I_Contact( "DATOS_PRODUCCION_MODO_A".flag_brazo2_extracción_superior )
      R_Coil( "DATOS_PRODUCCION".flag_brazo2_extracción_superior )
   END_RUNG
   RUNG wire#w1
      Contact( "DATOS_PRODUCCION_MODO_A".flag_sentido_cinta_inferior )
      S_Coil( "DATOS_PRODUCCION".flag_sentido_cinta_inferior )
   END_RUNG
   RUNG wire#w1
      I_Contact( "DATOS_PRODUCCION_MODO_A".flag_sentido_cinta_inferior )
      R_Coil( "DATOS_PRODUCCION".flag_sentido_cinta_inferior )
   END_RUNG
   RUNG wire#w1
      Contact( "DATOS_PRODUCCION_MODO_A".flag_sentido_cinta_superior )
      S_Coil( "DATOS_PRODUCCION".flag_sentido_cinta_superior )
   END_RUNG
   RUNG wire#w1
      I_Contact( "DATOS_PRODUCCION_MODO_A".flag_sentido_cinta_superior )
      R_Coil( "DATOS_PRODUCCION".flag_sentido_cinta_superior )
   END_RUNG
   // the same network as SCL:
   IF "XA" THEN
       "DATOS_PRODUCCION".temp_referencia_laminado := "DATOS_PRODUCCION_MODO_A".temp_ref_laminado;
   END_IF;
   IF "XA" AND "DATOS_PRODUCCION_MODO_A".flag_brazo1_alimentar THEN
       "DATOS_PRODUCCION".flag_brazo1_alimentar := TRUE;
   END_IF;
   IF "XA" AND NOT "DATOS_PRODUCCION_MODO_A".flag_brazo1_alimentar THEN
       "DATOS_PRODUCCION".flag_brazo1_alimentar := FALSE;
   END_IF;
   IF "XA" AND "DATOS_PRODUCCION_MODO_A".flag_brazo1_extracción_inferior THEN
       "DATOS_PRODUCCION".flag_brazo1_extracción_inferior := TRUE;
   END_IF;
   IF "XA" AND NOT "DATOS_PRODUCCION_MODO_A".flag_brazo1_extracción_inferior THEN
       "DATOS_PRODUCCION".flag_brazo1_extracción_inferior := FALSE;
   END_IF;
   IF "XA" AND "DATOS_PRODUCCION_MODO_A".flag_brazo1_extracción_superior THEN
       "DATOS_PRODUCCION".flag_brazo1_extracción_superior := TRUE;
   END_IF;
   IF "XA" AND NOT "DATOS_PRODUCCION_MODO_A".flag_brazo1_extracción_superior THEN
       "DATOS_PRODUCCION".flag_brazo1_extracción_superior := FALSE;
   END_IF;
   IF "XA" AND "DATOS_PRODUCCION_MODO_A".flag_brazo2_alimentar THEN
       "DATOS_PRODUCCION".flag_brazo2_alimentar := TRUE;
   END_IF;
   IF "XA" AND NOT "DATOS_PRODUCCION_MODO_A".flag_brazo2_alimentar THEN
       "DATOS_PRODUCCION".flag_brazo2_alimentar := FALSE;
   END_IF;
   IF "XA" AND "DATOS_PRODUCCION_MODO_A".flag_brazo2_extracción_inferior THEN
       "DATOS_PRODUCCION".flag_brazo2_extracción_inferior := TRUE;
   END_IF;
   IF "XA" AND NOT "DATOS_PRODUCCION_MODO_A".flag_brazo2_extracción_inferior THEN
       "DATOS_PRODUCCION".flag_brazo2_extracción_inferior := FALSE;
   END_IF;
   IF "XA" AND "DATOS_PRODUCCION_MODO_A".flag_brazo2_extracción_superior THEN
       "DATOS_PRODUCCION".flag_brazo2_extracción_superior := TRUE;
   END_IF;
   IF "XA" AND NOT "DATOS_PRODUCCION_MODO_A".flag_brazo2_extracción_superior THEN
       "DATOS_PRODUCCION".flag_brazo2_extracción_superior := FALSE;
   END_IF;
   IF "XA" AND "DATOS_PRODUCCION_MODO_A".flag_sentido_cinta_inferior THEN
       "DATOS_PRODUCCION".flag_sentido_cinta_inferior := TRUE;
   END_IF;
   IF "XA" AND NOT "DATOS_PRODUCCION_MODO_A".flag_sentido_cinta_inferior THEN
       "DATOS_PRODUCCION".flag_sentido_cinta_inferior := FALSE;
   END_IF;
   IF "XA" AND "DATOS_PRODUCCION_MODO_A".flag_sentido_cinta_superior THEN
       "DATOS_PRODUCCION".flag_sentido_cinta_superior := TRUE;
   END_IF;
   IF "XA" AND NOT "DATOS_PRODUCCION_MODO_A".flag_sentido_cinta_superior THEN
       "DATOS_PRODUCCION".flag_sentido_cinta_superior := FALSE;
   END_IF;
END_REGION

REGION Network 2: Tratamiento Modo de Marcha B
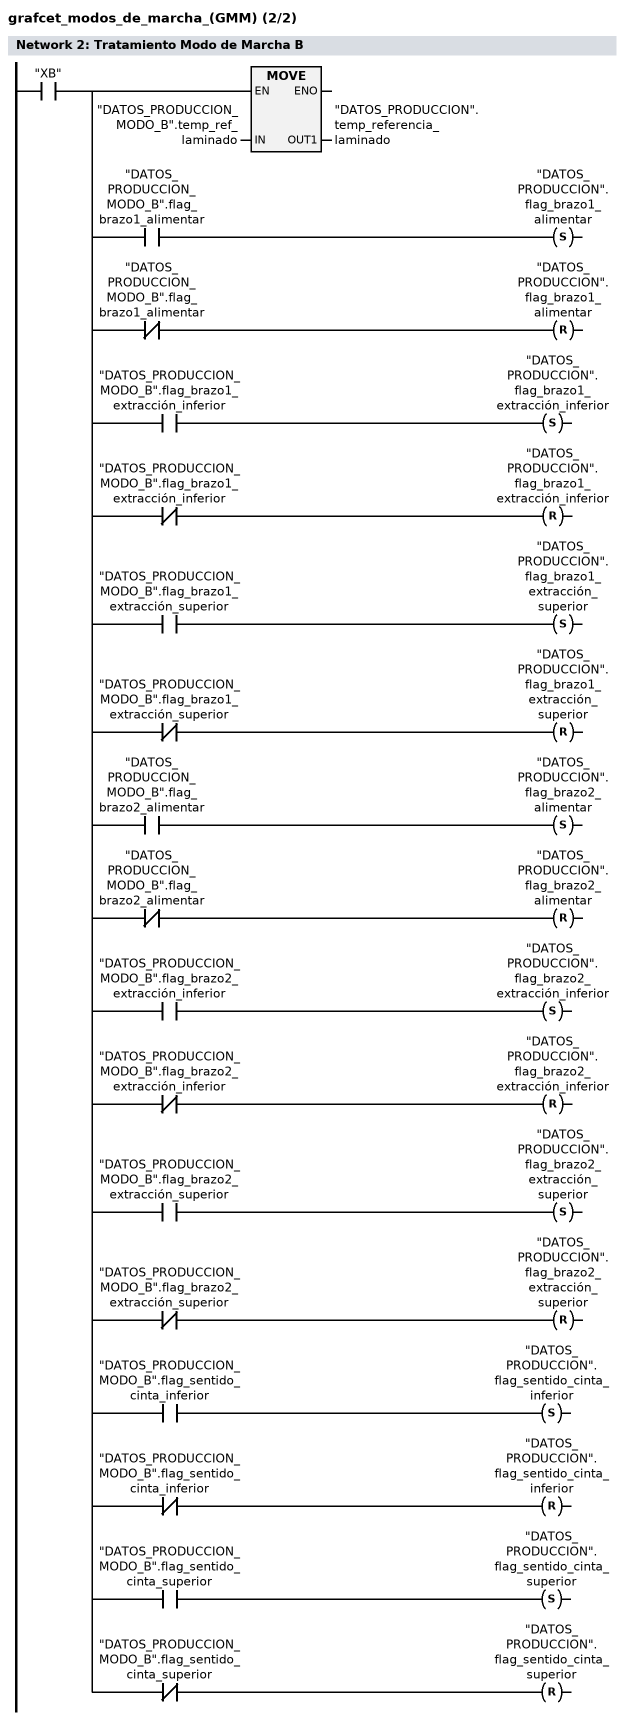
   RUNG wire#powerrail
      Contact( "XB" )
      wire#w1
      Move(in := "DATOS_PRODUCCION_MODO_B".temp_ref_laminado, out1 => "DATOS_PRODUCCION".temp_referencia_laminado)
   END_RUNG
   RUNG wire#w1
      Contact( "DATOS_PRODUCCION_MODO_B".flag_brazo1_alimentar )
      S_Coil( "DATOS_PRODUCCION".flag_brazo1_alimentar )
   END_RUNG
   RUNG wire#w1
      I_Contact( "DATOS_PRODUCCION_MODO_B".flag_brazo1_alimentar )
      R_Coil( "DATOS_PRODUCCION".flag_brazo1_alimentar )
   END_RUNG
   RUNG wire#w1
      Contact( "DATOS_PRODUCCION_MODO_B".flag_brazo1_extracción_inferior )
      S_Coil( "DATOS_PRODUCCION".flag_brazo1_extracción_inferior )
   END_RUNG
   RUNG wire#w1
      I_Contact( "DATOS_PRODUCCION_MODO_B".flag_brazo1_extracción_inferior )
      R_Coil( "DATOS_PRODUCCION".flag_brazo1_extracción_inferior )
   END_RUNG
   RUNG wire#w1
      Contact( "DATOS_PRODUCCION_MODO_B".flag_brazo1_extracción_superior )
      S_Coil( "DATOS_PRODUCCION".flag_brazo1_extracción_superior )
   END_RUNG
   RUNG wire#w1
      I_Contact( "DATOS_PRODUCCION_MODO_B".flag_brazo1_extracción_superior )
      R_Coil( "DATOS_PRODUCCION".flag_brazo1_extracción_superior )
   END_RUNG
   RUNG wire#w1
      Contact( "DATOS_PRODUCCION_MODO_B".flag_brazo2_alimentar )
      S_Coil( "DATOS_PRODUCCION".flag_brazo2_alimentar )
   END_RUNG
   RUNG wire#w1
      I_Contact( "DATOS_PRODUCCION_MODO_B".flag_brazo2_alimentar )
      R_Coil( "DATOS_PRODUCCION".flag_brazo2_alimentar )
   END_RUNG
   RUNG wire#w1
      Contact( "DATOS_PRODUCCION_MODO_B".flag_brazo2_extracción_inferior )
      S_Coil( "DATOS_PRODUCCION".flag_brazo2_extracción_inferior )
   END_RUNG
   RUNG wire#w1
      I_Contact( "DATOS_PRODUCCION_MODO_B".flag_brazo2_extracción_inferior )
      R_Coil( "DATOS_PRODUCCION".flag_brazo2_extracción_inferior )
   END_RUNG
   RUNG wire#w1
      Contact( "DATOS_PRODUCCION_MODO_B".flag_brazo2_extracción_superior )
      S_Coil( "DATOS_PRODUCCION".flag_brazo2_extracción_superior )
   END_RUNG
   RUNG wire#w1
      I_Contact( "DATOS_PRODUCCION_MODO_B".flag_brazo2_extracción_superior )
      R_Coil( "DATOS_PRODUCCION".flag_brazo2_extracción_superior )
   END_RUNG
   RUNG wire#w1
      Contact( "DATOS_PRODUCCION_MODO_B".flag_sentido_cinta_inferior )
      S_Coil( "DATOS_PRODUCCION".flag_sentido_cinta_inferior )
   END_RUNG
   RUNG wire#w1
      I_Contact( "DATOS_PRODUCCION_MODO_B".flag_sentido_cinta_inferior )
      R_Coil( "DATOS_PRODUCCION".flag_sentido_cinta_inferior )
   END_RUNG
   RUNG wire#w1
      Contact( "DATOS_PRODUCCION_MODO_B".flag_sentido_cinta_superior )
      S_Coil( "DATOS_PRODUCCION".flag_sentido_cinta_superior )
   END_RUNG
   RUNG wire#w1
      I_Contact( "DATOS_PRODUCCION_MODO_B".flag_sentido_cinta_superior )
      R_Coil( "DATOS_PRODUCCION".flag_sentido_cinta_superior )
   END_RUNG
   // the same network as SCL:
   IF "XB" THEN
       "DATOS_PRODUCCION".temp_referencia_laminado := "DATOS_PRODUCCION_MODO_B".temp_ref_laminado;
   END_IF;
   IF "XB" AND "DATOS_PRODUCCION_MODO_B".flag_brazo1_alimentar THEN
       "DATOS_PRODUCCION".flag_brazo1_alimentar := TRUE;
   END_IF;
   IF "XB" AND NOT "DATOS_PRODUCCION_MODO_B".flag_brazo1_alimentar THEN
       "DATOS_PRODUCCION".flag_brazo1_alimentar := FALSE;
   END_IF;
   IF "XB" AND "DATOS_PRODUCCION_MODO_B".flag_brazo1_extracción_inferior THEN
       "DATOS_PRODUCCION".flag_brazo1_extracción_inferior := TRUE;
   END_IF;
   IF "XB" AND NOT "DATOS_PRODUCCION_MODO_B".flag_brazo1_extracción_inferior THEN
       "DATOS_PRODUCCION".flag_brazo1_extracción_inferior := FALSE;
   END_IF;
   IF "XB" AND "DATOS_PRODUCCION_MODO_B".flag_brazo1_extracción_superior THEN
       "DATOS_PRODUCCION".flag_brazo1_extracción_superior := TRUE;
   END_IF;
   IF "XB" AND NOT "DATOS_PRODUCCION_MODO_B".flag_brazo1_extracción_superior THEN
       "DATOS_PRODUCCION".flag_brazo1_extracción_superior := FALSE;
   END_IF;
   IF "XB" AND "DATOS_PRODUCCION_MODO_B".flag_brazo2_alimentar THEN
       "DATOS_PRODUCCION".flag_brazo2_alimentar := TRUE;
   END_IF;
   IF "XB" AND NOT "DATOS_PRODUCCION_MODO_B".flag_brazo2_alimentar THEN
       "DATOS_PRODUCCION".flag_brazo2_alimentar := FALSE;
   END_IF;
   IF "XB" AND "DATOS_PRODUCCION_MODO_B".flag_brazo2_extracción_inferior THEN
       "DATOS_PRODUCCION".flag_brazo2_extracción_inferior := TRUE;
   END_IF;
   IF "XB" AND NOT "DATOS_PRODUCCION_MODO_B".flag_brazo2_extracción_inferior THEN
       "DATOS_PRODUCCION".flag_brazo2_extracción_inferior := FALSE;
   END_IF;
   IF "XB" AND "DATOS_PRODUCCION_MODO_B".flag_brazo2_extracción_superior THEN
       "DATOS_PRODUCCION".flag_brazo2_extracción_superior := TRUE;
   END_IF;
   IF "XB" AND NOT "DATOS_PRODUCCION_MODO_B".flag_brazo2_extracción_superior THEN
       "DATOS_PRODUCCION".flag_brazo2_extracción_superior := FALSE;
   END_IF;
   IF "XB" AND "DATOS_PRODUCCION_MODO_B".flag_sentido_cinta_inferior THEN
       "DATOS_PRODUCCION".flag_sentido_cinta_inferior := TRUE;
   END_IF;
   IF "XB" AND NOT "DATOS_PRODUCCION_MODO_B".flag_sentido_cinta_inferior THEN
       "DATOS_PRODUCCION".flag_sentido_cinta_inferior := FALSE;
   END_IF;
   IF "XB" AND "DATOS_PRODUCCION_MODO_B".flag_sentido_cinta_superior THEN
       "DATOS_PRODUCCION".flag_sentido_cinta_superior := TRUE;
   END_IF;
   IF "XB" AND NOT "DATOS_PRODUCCION_MODO_B".flag_sentido_cinta_superior THEN
       "DATOS_PRODUCCION".flag_sentido_cinta_superior := FALSE;
   END_IF;
END_REGION

REGION Network 3 (STL): X10->XA
   // Para implementar el forzado de EMER, se ha incluido el estado de emergencia "X21" negado
         A     "X10";
         AN    "X21";
         A     "MA";
         R     "X10";
         S     "XA";
END_REGION

REGION Network 4 (STL): XA->X10
         A     "XA";
         AN    "MA";
         R     "XA";
         S     "X10";
END_REGION

REGION Network 5 (STL): X10->XB
   // Para implementar el forzado de EMER, se ha incluido el estado de emergencia "X21" negado
         A     "X10";
         AN    "X21";
         A     "MB";
         R     "X10";
         S     "XB";
END_REGION

REGION Network 6 (STL): XB->X10
         A     "XB";
         AN    "MB";
         R     "XB";
         S     "X10";
END_REGION
END_FUNCTION

FUNCTION "grafcet_marcha_y_parada_controlada_(GMPC)" : Void   // FC12, LAD
TITLE = Grafcet de Marcha y Parada Controlada
{ S7_Optimized_Access := 'TRUE' }
VERSION : 0.1
// Se coordina con el grafcet de producción para lograr una parada controlada dentro del tiempo establecido
   VAR_TEMP
      disparo_temp_parada_controlada : Bool;
   END_VAR
BEGIN

REGION Network 1 (STL): XOFF->XON
   // Se ha incluido como condición "X21" negada para implementar el forzado. Realmente no es necesario, ya que durante el defecto por emergencia "X0" será ==FALSE. Además, deberá haber un modo de marcha activo.
         A     "XOFF";
         A(;
         O     "XA";
         O     "XB";
         );
         AN    "X21";
         A     "X0";
         A     "mpON";
         AN    "OFF";
         R     "XOFF";
         S     "XON";
END_REGION

REGION Network 2 (STL): XON->XOFF
         A     "XON";
         A     "OFF";
         R     "XON";
         S     "XOFF";
END_REGION

REGION Network 3 (STL): Gestión Señal de Disparo del Temporizador
   // Para evitar que el temporizador se dispare durante la emergencia.
         A     "X_Trabajo";
         A     "XOFF";
         =     #disparo_temp_parada_controlada;
END_REGION

REGION Network 4 (STL): Gestión Temporizador para la Parada Controlada
   // Se usará la salida del temporizador en el grafcet de producción GP para gestionar la parada controlada del sistema.
         CALL  TON, "TON_PARADA_Controlada_DB"
         ( IN := #disparo_temp_parada_controlada,
           PT := "DATOS_PRODUCCION".tiempo_parada_controlada,
           Q  := ,
           ET :=
         );
END_REGION
END_FUNCTION

// folder: Máquinas

FUNCTION_BLOCK "CNC (Corte/Serigrafía)"   // FB2, LAD
TITLE = Bloque Máquina (para las CNCs de corte y serigrafía)
{ S7_Optimized_Access := 'TRUE' }
VERSION : 0.1
// Incluye estados de defecto por tiempo límite, mal arranque y  emergencia. Se ha considerado una única señal de rearme que devuelve a la máquina al reposo desde la emergencia. Para volver desde el defecto se ha configurado un aviso que puede ser desactivado por el usuario (una vez se ha solucionado el problema).
// (BLOQUE AUTOCONTENIDO)
   VAR_INPUT
      Start : Bool;   // Señal de arranque de la máquina
      EMER : Bool;   // Señal de emergencia
      SE : Bool;   // Sensor de presencia a la entrada de la máquina
      máquina_en_posición : Bool;   // Aviso de que la máquina está posicionada adecuadamente para el arranque (tras solventarse un defecto, por ejemplo)
      Rearme : Bool;   // Señal de rearme de la máquina
      tiempo_límite : Time;   // Tiempo límite para completar la operación
   END_VAR
   VAR_OUTPUT
      MÁQUINA_ON : Bool;   // Actuador que representa el funcionamiento global de la máquina
      aviso_standby : Bool;   // Aviso de que la máquina está en standby
   END_VAR
   VAR_IN_OUT
      aviso_defecto : Bool;
   END_VAR
   VAR
      bit_de_trabajo : Bool;   // bit de trabajo para el arranque
      X_Standby : Bool;   // Estado de Standby
      X_Defecto_Tiempo : Bool;   // Estado de defecto de tiempo
      X_Defecto_Emergencia : Bool;   // Estado de defecto por emergencia
      X_Defecto_Posición : Bool;   // Estado de defecto por mal posicionamiento inicial
      X_Trabajo1 : Bool;   // Estado de trabajo de la máquina
      X_Trabajo2 : Bool;   // Estado anti-fugacidad
      M_flanco_rearme : Bool;   // Marca de flanco de la señal rearme
      M_flanco_defecto : Bool;   // Marca de flanco para el aviso de defecto
      temporizador : TON_TIME;
   END_VAR
   VAR_TEMP
      señal_temp : Bool;
   END_VAR
   VAR_TEMP   // added for the SCL form of the ladder/FBD networks
      _w1 : Bool;
   END_VAR
BEGIN

REGION Network 1 (STL): DESCONEXIÓN (Start:=False)
   // Aagado de la máquina, máxima prioridad. Se llama a las maniobras con RESET:=TRUE (en caso de haberlas).
   // Tan solo se ponen a cero las salidas, los estados internos se inicializarán en el arranque.
         AN    #Start;
         JCN   _RESET;
         CALL  RESET_TIMER
         ( "TIMER" := #temporizador
         );
         AN    #Start;
         R     #bit_de_trabajo;
         R     #aviso_standby;
         R     #MÁQUINA_ON;
         R     #aviso_defecto;
         BEC;
   _RESET:NOP   0;
END_REGION

REGION Network 2 (STL): DEFECTO (emergencia)
   // Defecto prioritario. LLamamos a las maniobras con RESET:=TRUE (en caso de haberlas)
         A     #EMER;
         S     #X_Defecto_Emergencia;
         R     #X_Standby;
         R     #X_Defecto_Tiempo;
         R     #X_Defecto_Posición;
         R     #X_Trabajo1;
END_REGION

REGION Network 3 (STL): DEFECTO (tiempo excedido durante la expansión)
   // Ante el aviso de defecto por tiempo (lo proporciona el bloque maniobra) se accede al estado de defecto.
         A     #X_Trabajo1;
         A     #temporizador.Q;
         S     #X_Defecto_Tiempo;
         R     #X_Trabajo1;
END_REGION

REGION Network 4 (STL): DEFECTO (mal posicionamiento en el arranque)
   // Si al arrancar, la máquina no está posicionada correctamente, se accede al correspondiente estado de defecto.
         A     #X_Standby;
         AN    #máquina_en_posición;
         S     #X_Defecto_Posición;
         R     #X_Standby;
END_REGION

REGION Network 5 (STL): Aviso de defecto (para el rearme)
   // Se avisará al usuario cuando la máquina haya entrado en defecto
         A     #X_Defecto_Posición;
         O     #X_Defecto_Tiempo;
         FP    #M_flanco_defecto;
         S     #aviso_defecto;
END_REGION

REGION Network 6 (STL): REARME (emergencia)
   // Una vez se ha solucionado el problema  se vuelve al reposo con el flanco positivo de la señal rearme.
         A     #Rearme;
         FP    #M_flanco_rearme;
         A     #X_Defecto_Emergencia;
         AN    #EMER;
         S     #X_Standby;
         R     #X_Defecto_Emergencia;
END_REGION

REGION Network 7: REARME (Defecto de tiempo o posición)
   // Una vez se ha solucionado el problema, se vuelve al reposo al desactivarse el aviso de error (por el usuario)
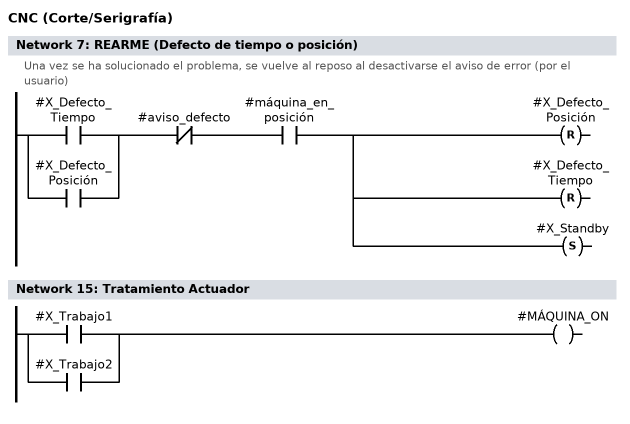
   RUNG wire#powerrail
      Contact( #X_Defecto_Tiempo )
      wire#w1
      I_Contact( #aviso_defecto )
      Contact( #máquina_en_posición )
      wire#w2
      R_Coil( #X_Defecto_Posición )
   END_RUNG
   RUNG wire#powerrail
      Contact( #X_Defecto_Posición )
   END_RUNG wire#w1
   RUNG wire#w2
      R_Coil( #X_Defecto_Tiempo )
   END_RUNG
   RUNG wire#w2
      S_Coil( #X_Standby )
   END_RUNG
   // the same network as SCL:
   #_w1 := (#X_Defecto_Tiempo OR #X_Defecto_Posición) AND NOT #aviso_defecto AND #máquina_en_posición;
   IF #_w1 THEN
       #X_Defecto_Posición := FALSE;
       #X_Defecto_Tiempo := FALSE;
       #X_Standby := TRUE;
   END_IF;
END_REGION

REGION Network 8 (STL): ARRANQUE
   // Arrancamos la máquina, inicializando el estado de standby (X0)
         A     #Start;
         FP    #bit_de_trabajo;
         S     #X_Standby;
         R     #X_Defecto_Tiempo;
         R     #X_Defecto_Emergencia;
         R     #X_Defecto_Posición;
         R     #M_flanco_defecto;
         R     #M_flanco_rearme;
         R     #X_Trabajo1;
         R     #X_Trabajo2;
END_REGION

REGION Network 9 (STL): Configuración señal temporizador
         A     #X_Trabajo1;
         O     #X_Trabajo2;
         =     #señal_temp;
END_REGION

REGION Network 10 (STL): Configuración Temporizador
   // Se empleará un TON (sin memoria)
         CALL  #temporizador
         ( IN := #señal_temp,
           PT := #tiempo_límite,
           Q  := ,
           ET :=
         );
END_REGION

REGION Network 11 (STL): X_Standby -> X_Trabajo1
   // La máquina comienza el tratamiento cuando detecta que se le ha pasado una pieza.
         A     #X_Standby;
         A     #SE;
         A     #máquina_en_posición;
         R     #X_Standby;
         S     #X_Trabajo1;
END_REGION

REGION Network 12 (STL): X_Trabajo1->X_Trabajo2
   // Estado anti-fugaz
         A     #X_Trabajo1;
         AN    #máquina_en_posición;
         R     #X_Trabajo1;
         S     #X_Trabajo2;
END_REGION

REGION Network 13 (STL): X_Trabajo2 -> X_Standby
   // Vuelta al estado de standby al terminar la operación de tratamiento de la pieza y estar la máquina posicionada.
         A     #X_Trabajo2;
         A     #máquina_en_posición;
         R     #X_Trabajo2;
         S     #X_Standby;
END_REGION

REGION Network 14 (STL): Aviso de Standby (para el usuario)
   // Avisa de que la máquina está en standby y funcionando correctamente
         A     #X_Standby;
         =     #aviso_standby;
END_REGION

REGION Network 15: Tratamiento Actuador
   RUNG wire#powerrail
      Contact( #X_Trabajo1 )
      wire#w1
      Coil( #MÁQUINA_ON )
   END_RUNG
   RUNG wire#powerrail
      Contact( #X_Trabajo2 )
   END_RUNG wire#w1
   // the same network as SCL:
   #MÁQUINA_ON := #X_Trabajo1 OR #X_Trabajo2;
END_REGION
END_FUNCTION_BLOCK

FUNCTION_BLOCK "Pistón (Máquina)"   // FB4, LAD
TITLE = Bloque Máquina (pistón con ciclo expansión-compresión)
{ S7_Optimized_Access := 'TRUE' }
VERSION : 0.1
// Incluye estados de defecto por tiempo límite, mal arranque y por emergencia. Se ha considerado una única señal de rearme que devuelve a la máquina al reposo desde la emergencia. Para volver desde el defecto se ha configurado un aviso que puede ser desactivado por el usuario (una vez se ha solucionado el problema).
// (BLOQUE AUTOCONTENIDO)
// (EMPLEA MANIOBRAS)
   VAR_INPUT
      Start : Bool;   // Señal de arranque de la máquina
      EMER : Bool;   // Señal de emergencia
      SC : Bool;   // Fin de carrera (pistón comprimido)
      SE : Bool;   // Fin de carreara (pistón expandido)
      Rearme : Bool;   // Señal de rearme de la máquina
      pieza_detectada : Bool;   // Aviso del sensor de presencia de que hay una pieza frente al pistón
      pieza_válida : Bool;   // Aviso del lector de código, que indica si la pieza que se aproxima deberá ser incorporada
      tiempo_expansión : Time;   // Tiempo límite para completar la maniobra de expansión
      tiempo_compresión : Time;   // Tiempo límite para completar la maniobra de compresión
      aviso_CNC_disponible : Bool;   // Aviso de que la máquina que se desea alimentar está disponible (en standby)
   END_VAR
   VAR_OUTPUT
      EXP : Bool;   // Actuador que expande el cilindro
      COMP : Bool;   // Actuador que comprime el pistón
      aviso_standby : Bool;   // Aviso de que la máquina está en standby
   END_VAR
   VAR_IN_OUT
      aviso_defecto : Bool;
   END_VAR
   VAR
      bit_de_trabajo : Bool;   // bit de trabajo para el arranque
      X0 : Bool;   // Estado de Standby
      X1 : Bool;   // Estado de Expansión
      X2 : Bool;   // Estado de Compresión
      X3 : Bool;   // Estado de defecto por exceso de tiempo
      X4 : Bool;   // Estado de defecto por emergencia
      X5 : Bool;   // Estado de defecto por mal arranque
      M_flanco_rearme : Bool;   // Marca de flanco para la señal rearme
      Pistón_Expansión : "Pistón (Maniobra Simple)";
      expansión_no_ok : Bool;   // Aviso de que el cilindro no se ha expandido en el tiempo especificado
      expansión_ok : Bool;   // Aviso de que la expansión se ha completado
      Pistón_Compresión : "Pistón (Maniobra Simple)";
      compresión_no_ok : Bool;   // Aviso de que la compresión se ha completado con éxito
      compresión_ok : Bool;   // Aviso de que la compresión no se ha completado en el tiempo especificado
      M_flanco_defecto : Bool;   // Marca de flanco para el aviso de defecto
      M_flanco_pieza_detectada : Bool;   // Marca de flanco de la señal pieza_detectada
   END_VAR
   VAR_TEMP
      M_pulso_rearme : Bool;
      M_pulso_pieza_detectada : Bool;
   END_VAR
   VAR_TEMP   // added for the SCL form of the ladder/FBD networks
      _w1 : Bool;
   END_VAR
BEGIN

REGION Network 1 (STL): DESCONEXIÓN (Start:=False)
   // Aagado de la máquina, máxima prioridad. Se llama a las maniobras con RESET:=TRUE.
   // Tan solo se ponen a cero las salidas, los estados internos se inicializarán en el arranque.
         AN    #Start;
         JCN   _OFF;
         CALL  #Pistón_Compresión
         ( SFIN                      := ,
           tiempo_limite             := ,
           RESET                     := TRUE,
           ACT                       := #COMP,
           aviso_error_tiempo_limite := #compresión_no_ok,
           aviso_fin_maniobra        := #compresión_ok
         );
         CALL  #Pistón_Expansión
         ( SFIN                      := ,
           tiempo_limite             := ,
           RESET                     := TRUE,
           ACT                       := #EXP,
           aviso_error_tiempo_limite := #compresión_no_ok,
           aviso_fin_maniobra        := #compresión_ok
         );
         AN    #Start;
         R     #bit_de_trabajo;
         R     #aviso_standby;
         R     #aviso_defecto;
         BEC;
   _OFF: NOP   0;
END_REGION

REGION Network 2 (STL): DEFECTO (emergencia)
   // Defecto prioritario. LLamamos a las maniobras con RESET:=TRUE
         A     #EMER;
         JCN   _EMER;
         CALL  #Pistón_Compresión
         ( SFIN                      := ,
           tiempo_limite             := ,
           RESET                     := TRUE,
           ACT                       := #COMP,
           aviso_error_tiempo_limite := #compresión_no_ok,
           aviso_fin_maniobra        := #compresión_ok
         );
         CALL  #Pistón_Expansión
         ( SFIN                      := ,
           tiempo_limite             := ,
           RESET                     := TRUE,
           ACT                       := #EXP,
           aviso_error_tiempo_limite := #expansión_no_ok,
           aviso_fin_maniobra        := #expansión_ok
         );
         A     #EMER;
         S     #X4;
         R     #X0;
         R     #X1;
         R     #X2;
         R     #X3;
         R     #X5;
   _EMER:NOP   0;
END_REGION

REGION Network 3 (STL): DEFECTO (mal arranque)
   // Si al arrancar el fin de carrera de pistón comprimido no está activado, se accede a este estado de defecto.
         A     #X0;
         AN    #SC;
         R     #X0;
         S     #X5;
END_REGION

REGION Network 4 (STL): DEFECTO (tiempo excedido durante la expansión)
   // Ante el aviso de defecto por tiempo (lo proporciona el bloque maniobra) se accede al estado de defecto.
         A     #X1;
         A     #expansión_no_ok;
         S     #X3;
         R     #X1;
END_REGION

REGION Network 5 (STL): DEFECTO (tiempo excedido durante la compresión)
   // Ante el aviso de defecto por tiempo (lo proporciona el bloque maniobra) se accede al estado de defecto.
         A     #X2;
         A     #compresión_no_ok;
         R     #X2;
         S     #X3;
END_REGION

REGION Network 6 (STL): Flanco de la señal Rearme
   // La señal rearme, que devuelve al sistema al reposo desde cuelquier defecto, funciona por flanco positivo.
         A     #Rearme;
         FP    #M_flanco_rearme;
         =     #M_pulso_rearme;
END_REGION

REGION Network 7 (STL): REARME (emergencia)
   // Una vez se ha solucionado el problema (comprobación con SC) se vuelve al reposo con el flanco positivo de la señal rearme.
         A     #X4;
         AN    #EMER;
         A     #M_pulso_rearme;
         R     #X4;
         S     #X0;
END_REGION

REGION Network 8: REARME (Defecto de mal arranque o tiempo)
   // Una vez se ha solucionado el problema se vuelve al reposo al desactivarse el aviso de error (por el usuario)
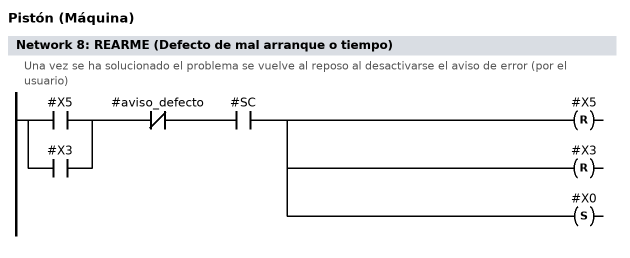
   RUNG wire#powerrail
      Contact( #X5 )
      wire#w1
      I_Contact( #aviso_defecto )
      Contact( #SC )
      wire#w2
      R_Coil( #X5 )
   END_RUNG
   RUNG wire#powerrail
      Contact( #X3 )
   END_RUNG wire#w1
   RUNG wire#w2
      R_Coil( #X3 )
   END_RUNG
   RUNG wire#w2
      S_Coil( #X0 )
   END_RUNG
   // the same network as SCL:
   #_w1 := (#X5 OR #X3) AND NOT #aviso_defecto AND #SC;
   IF #_w1 THEN
       #X5 := FALSE;
       #X3 := FALSE;
       #X0 := TRUE;
   END_IF;
END_REGION

REGION Network 9 (STL): Arranque
   // Arrancamos la máquina, inicializando el estado de standby (X0)
         A     #Start;
         FP    #bit_de_trabajo;
         S     #X0;
         R     #X1;
         R     #X2;
         R     #X3;
         R     #X3;
         R     #X4;
         R     #X5;
         R     #M_flanco_defecto;
         R     #M_flanco_rearme;
         R     #M_flanco_pieza_detectada;
END_REGION

REGION Network 10 (STL): Flanco de la señal pieza_detectada
         A     #pieza_detectada;
         FP    #M_flanco_pieza_detectada;
         =     #M_pulso_pieza_detectada;
END_REGION

REGION Network 11 (STL): X0 -> X1
   // Detección de pieza
         A     #X0;
         A     #SC;
         A     #M_pulso_pieza_detectada;
         A     #pieza_válida;
         A     #aviso_CNC_disponible;
         R     #X0;
         S     #X1;
END_REGION

REGION Network 12 (STL): X1->X2 (Maniobra de expansión)
   // LLamada a la maniobra y transición si ésta se completa dentro del tiempo especificado.
         A     #X1;
         JCN   _EXP;
         CALL  #Pistón_Expansión
         ( SFIN                      := #SE,
           tiempo_limite             := #tiempo_expansión,
           RESET                     := FALSE,
           ACT                       := #EXP,
           aviso_error_tiempo_limite := #expansión_no_ok,
           aviso_fin_maniobra        := #expansión_ok
         );
         A     #X1;
         A     #expansión_ok;
         R     #X1;
         S     #X2;
   _EXP: NOP   0;
END_REGION

REGION Network 13 (STL): X2->X0 (Maniobra de compresión)
   // LLamada a la maniobra y vuelta al reposo si ésta se completa dentro del tiempo especificado.
         A     #X2;
         JCN   _COMP;
         CALL  #Pistón_Compresión
         ( SFIN                      := #SC,
           tiempo_limite             := #tiempo_compresión,
           RESET                     := FALSE,
           ACT                       := #COMP,
           aviso_error_tiempo_limite := #compresión_no_ok,
           aviso_fin_maniobra        := #compresión_ok
         );
         A     #X2;
         A     #compresión_ok;
         R     #X2;
         S     #X0;
   _COMP:NOP   0;
END_REGION

REGION Network 14 (STL): Aviso de defecto (para el rearme)
   // Se avisará al usuario cuando la máquina haya entrado en defecto
         A     #X3;
         O     #X5;
         FP    #M_flanco_defecto;
         S     #aviso_defecto;
END_REGION

REGION Network 15 (STL): Aviso de Standby (para el usuario)
   // Avisa de que la máquina está en standby y funcionando correctamente
         A     #X0;
         =     #aviso_standby;
END_REGION
END_FUNCTION_BLOCK

FUNCTION_BLOCK "CNC (Laminado)"   // FB5, LAD
TITLE = Bloque Máquina (para la CNCs de laminado)
{ S7_Optimized_Access := 'TRUE' }
VERSION : 0.1
// Incluye estados de defecto por tiempo límite, mal arranque, lectura incorrecta y  emergencia. Se ha considerado una única señal de rearme que devuelve a la máquina al reposo desde la emergencia. Para volver desde el defecto se ha configurado un aviso que puede ser desactivado por el usuario (una vez se ha solucionado el problema).
// (BLOQUE AUTOCONTENIDO)
   VAR_INPUT
      Start : Bool;   // Señal de arranque
      EMER : Bool;   // Señal de activación del estado de emergencia
      tiempo : Time;   // Tiempo límite para tratar la pieza
      máquina_en_posición : Bool;   // Aviso de que la máquina está posicionada adecuadamente para comenzar la operación de laminado
      Rearme : Bool;   // Señal de rearme (emergencia)
      error_lectura_piro : Bool;   // Aviso de lectura errónea del pirómetro
      SE : Bool;   // Sensor de presencia a laentrada de la máquina
      lectura_pirómetro : Real;   // Lectura del pirómetro en ºC
      T_ref : Real;   // Temperatura a la que se deseará mantener la pieza.
   END_VAR
   VAR_OUTPUT
      aviso_standby : Bool;   // Aviso de máquina en standby
      MÁQUINA_ON : Bool;   // Actuador que engloba el funcionamiento de la máquina
      LÁMPARA_IR_ON : Bool;   // Actuador que activa la lámpara IR
   END_VAR
   VAR_IN_OUT
      aviso_defecto : Bool;   // Aviso de defecto (de utilidad para el rearme)
   END_VAR
   VAR
      X_standby : Bool;   // Estado de espera
      X_trabajo1 : Bool;   // Estado de calentamiento y tratamientpo de la pieza
      X_trabajo2 : Bool;   // Estado anti-fugacidad
      X_defecto_tiempo : Bool;   // Estado de defecto por tiempo sobrepasado
      X_defecto_emergencia : Bool;   // Estado de defecto por emergencia
      X_defecto_lectura : Bool;   // Estado de defecto por lectura errónea
      X_defecto_posición : Bool;   // Estado de defecto por mal posicionamiento
      bit_de_trabajo : Bool;   // Bit de trabajo para el arranque
      M_flanco_rearme : Bool;   // Marca de flanco de la señal de rearme
      M_flanco_defecto : Bool;   // Marca de flanco del aviso de defecto
      temporizador : TON_TIME;   // TON para el defecto de tiempo
   END_VAR
   VAR_TEMP
      señal_temp : Bool;   // Señal de disparo del temporizador
   END_VAR
   VAR_TEMP   // added for the SCL form of the ladder/FBD networks
      _w1 : Bool;
   END_VAR
BEGIN

REGION Network 1 (STL): DESCONEXIÓN (Start:=False)
   // Aagado de la máquina, máxima prioridad. Se llama a las maniobras con RESET:=TRUE (en caso de haberlas).
   // Tan solo se ponen a cero las salidas, los estados internos se inicializarán en el arranque.
         AN    #Start;
         JCN   _RESET;
         CALL  RESET_TIMER
         ( "TIMER" := #temporizador
         );
         AN    #Start;
         R     #bit_de_trabajo;
         R     #aviso_standby;
         R     #MÁQUINA_ON;
         R     #aviso_defecto;
         R     #LÁMPARA_IR_ON;
         BEC;
   _RESET:NOP   0;
END_REGION

REGION Network 2 (STL): DEFECTO (emergencia)
   // Defecto prioritario. LLamamos a las maniobras con RESET:=TRUE (en caso de haberlas)
         A     #EMER;
         S     #X_defecto_emergencia;
         R     #X_standby;
         R     #X_defecto_lectura;
         R     #X_defecto_tiempo;
         R     #X_defecto_posición;
         R     #X_trabajo1;
END_REGION

REGION Network 3 (STL): DEFECTO (lectura incorrecta)
   // Máxima prioridad (después de la emergencia)
         A     #error_lectura_piro;
         AN    #X_defecto_emergencia;
         S     #X_defecto_lectura;
         R     #X_standby;
         R     #X_trabajo1;
         R     #X_defecto_posición;
         R     #X_defecto_tiempo;
END_REGION

REGION Network 4 (STL): DEFECTO (tiempo excedido)
   // Ante el aviso de defecto por tiempo se accede al estado de defecto.
         A     #X_trabajo1;
         A     #temporizador.Q;
         S     #X_defecto_tiempo;
         R     #X_trabajo1;
END_REGION

REGION Network 5 (STL): DEFECTO (mal posicionamiento en el arranque)
   // Si al arrancar, la máquina no está posicionada correctamente, se accede al correspondiente estado de defecto.
         A     #X_standby;
         AN    #máquina_en_posición;
         S     #X_defecto_posición;
         R     #X_standby;
END_REGION

REGION Network 6 (STL): Aviso de defecto (para el rearme)
   // Se avisará al usuario cuando la máquina haya entrado en defecto
         A     #X_defecto_posición;
         O     #X_defecto_tiempo;
         O     #X_defecto_lectura;
         FP    #M_flanco_defecto;
         S     #aviso_defecto;
END_REGION

REGION Network 7 (STL): REARME (emergencia)
   // Una vez se ha solucionado el problema  se vuelve al reposo con el flanco positivo de la señal rearme.
         A     #Rearme;
         FP    #M_flanco_rearme;
         A     #X_defecto_emergencia;
         AN    #EMER;
         S     #X_standby;
         R     #X_defecto_emergencia;
END_REGION

REGION Network 8: REARME (Defecto de tiempo o posición)
   // Una vez se ha solucionado el problema, se vuelve al reposo al desactivarse el aviso de error (por el usuario)
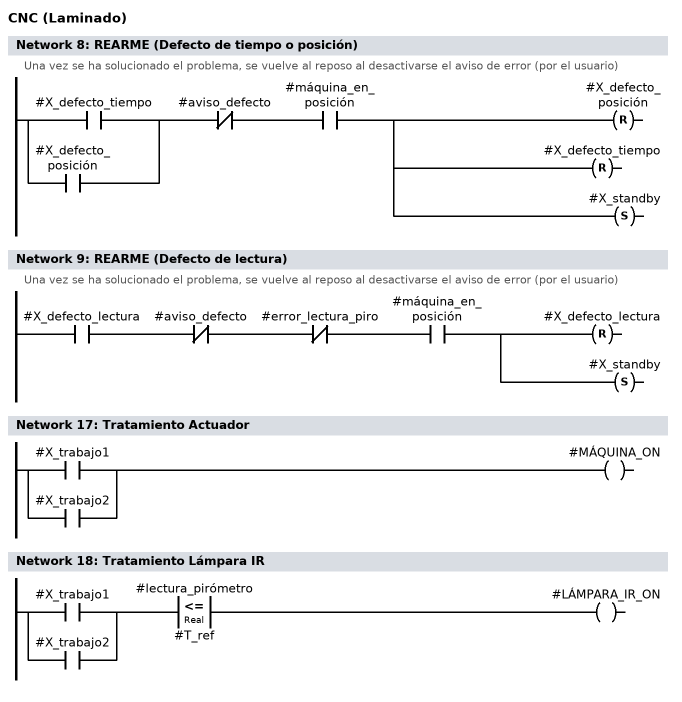
   RUNG wire#powerrail
      Contact( #X_defecto_tiempo )
      wire#w1
      I_Contact( #aviso_defecto )
      Contact( #máquina_en_posición )
      wire#w2
      R_Coil( #X_defecto_posición )
   END_RUNG
   RUNG wire#powerrail
      Contact( #X_defecto_posición )
   END_RUNG wire#w1
   RUNG wire#w2
      R_Coil( #X_defecto_tiempo )
   END_RUNG
   RUNG wire#w2
      S_Coil( #X_standby )
   END_RUNG
   // the same network as SCL:
   #_w1 := (#X_defecto_tiempo OR #X_defecto_posición) AND NOT #aviso_defecto AND #máquina_en_posición;
   IF #_w1 THEN
       #X_defecto_posición := FALSE;
       #X_defecto_tiempo := FALSE;
       #X_standby := TRUE;
   END_IF;
END_REGION

REGION Network 9: REARME (Defecto de lectura)
   // Una vez se ha solucionado el problema, se vuelve al reposo al desactivarse el aviso de error (por el usuario)
   RUNG wire#powerrail
      Contact( #X_defecto_lectura )
      I_Contact( #aviso_defecto )
      I_Contact( #error_lectura_piro )
      Contact( #máquina_en_posición )
      wire#w1
      R_Coil( #X_defecto_lectura )
   END_RUNG
   RUNG wire#w1
      S_Coil( #X_standby )
   END_RUNG
   // the same network as SCL:
   #_w1 := #X_defecto_lectura AND NOT #aviso_defecto AND NOT #error_lectura_piro AND #máquina_en_posición;
   IF #_w1 THEN
       #X_defecto_lectura := FALSE;
       #X_standby := TRUE;
   END_IF;
END_REGION

REGION Network 10 (STL): ARRANQUE
   // Arrancamos la máquina, inicializando el estado de standby (X0)
         A     #Start;
         FP    #bit_de_trabajo;
         S     #X_standby;
         R     #X_defecto_tiempo;
         R     #X_defecto_lectura;
         R     #X_defecto_emergencia;
         R     #X_defecto_posición;
         R     #M_flanco_defecto;
         R     #M_flanco_rearme;
         R     #X_trabajo1;
         R     #X_trabajo2;
END_REGION

REGION Network 11 (STL): Configuración Señal Temporizador
         A     #X_trabajo1;
         O     #X_trabajo2;
         =     #señal_temp;
END_REGION

REGION Network 12 (STL): Configuración Temporizador (tiempo límite)
   // Se empleará un TON (sin memoria)
         CALL  #temporizador
         ( IN := #señal_temp,
           PT := #tiempo,
           Q  := ,
           ET :=
         );
END_REGION

REGION Network 13 (STL): X_Standby -> X_Trabajo1
   // La máquina comienza el tratamiento cuando detecta que se le ha pasado una pieza.
         A     #X_standby;
         A     #SE;
         A     #máquina_en_posición;
         R     #X_standby;
         S     #X_trabajo1;
END_REGION

REGION Network 14 (STL): X_Trabajo1->X_Trabajo2
   // Para evitar que la etapa de trabajo pueda ser fugaz
         A     #X_trabajo1;
         AN    #máquina_en_posición;
         S     #X_trabajo2;
         R     #X_trabajo1;
END_REGION

REGION Network 15 (STL): X_Trabajo2 -> X_Standby
   // Vuelta al estado de standby al terminar la operación de tratamiento de la pieza y estar la máquina posicionada.
         A     #X_trabajo2;
         A     #máquina_en_posición;
         R     #X_trabajo2;
         S     #X_standby;
END_REGION

REGION Network 16 (STL): Aviso de Standby (para el usuario)
   // Avisa de que la máquina está en standby y funcionando correctamente
         A     #X_standby;
         =     #aviso_standby;
END_REGION

REGION Network 17: Tratamiento Actuador
   RUNG wire#powerrail
      Contact( #X_trabajo1 )
      wire#w1
      Coil( #MÁQUINA_ON )
   END_RUNG
   RUNG wire#powerrail
      Contact( #X_trabajo2 )
   END_RUNG wire#w1
   // the same network as SCL:
   #MÁQUINA_ON := #X_trabajo1 OR #X_trabajo2;
END_REGION

REGION Network 18: Tratamiento Lámpara IR
   RUNG wire#powerrail
      Contact( #X_trabajo1 )
      wire#w1
      { S7_Templates := "SrcType := Real" } LE_Contact(in1 := #lectura_pirómetro, in2 := #T_ref)
      Coil( #LÁMPARA_IR_ON )
   END_RUNG
   RUNG wire#powerrail
      Contact( #X_trabajo2 )
   END_RUNG wire#w1
   // the same network as SCL:
   #LÁMPARA_IR_ON := (#X_trabajo1 OR #X_trabajo2) AND (#lectura_pirómetro <= #T_ref);
END_REGION
END_FUNCTION_BLOCK

FUNCTION_BLOCK "Brazo de Carga/Descarga"   // FB6, LAD
TITLE = Bloque Máquina (para el Brazo de Carga/Descarga)
{ S7_Optimized_Access := 'TRUE' }
VERSION : 0.1
// 1. Incluye estados de defecto por tiempo límite, mal arranque y  emergencia. 
// 2. Se ha considerado una señal de rearme que devuelve a la máquina al reposo desde la emergencia. 
// 3. Para volver desde el defecto se ha configurado un aviso que puede ser desactivado por el usuario (una vez se ha solucionado el problema). 
// 4. Mediante el uso de "flags" se habilitarán las maniobras requeridas (carga, descarga superior y descarga inferior) en función del sentido de las cintas (modos de marcha).
// 5. Se han considerado las maniobras de alimentación por la cinta superior y descarga por las cintas superior e inferior. No se ha considerado la maniobra de alimentación por la cinta inferior (las máquinas se alimentan únicamente por arriba), aunque podría incorporarse fácilmente al bloque.
// (BLOQUE AUTOCONTENIDO)
   VAR_INPUT
      Start : Bool;   // Señal de arranque
      EMER : Bool;   // Señal de activación del estado de emergencia
      tiempo : Time;   // Tiempo límite para completar cualquiera de las maniobras
      brazo_en_posición : Bool;   // Aviso de que el brazo está posicionado adecuadamente para comenzar la siguiente maniobra
      Rearme : Bool;   // Señal de rearme (emergencia)
      S_superior : Bool;   // Sensor de presencia al inicio de la cinta superior para la detección de la llegada de piezas
      S_inferior : Bool;   // Sensor de presencia al inicio de la cinta inferior para la detección de la llegada de piezas
      fin_maniobra : Bool;   // Aviso de que la maniobra ha concluido
      orden_alimentar : Bool;   // Orden enviada por el sistema para comenzar la maniobra de alimentación
      flag_alim : Bool;   // "flag" que habilita la maniobra de alimentación (por la cinta superior)
      flag_extr_inf : Bool;   // "flag" que habilita la operación de extracción por la cinta inferior
      flag_extr_sup : Bool;   // "flag" que habilita la maniobra de extracción por la cinta superior
   END_VAR
   VAR_OUTPUT
      aviso_standby : Bool;   // Aviso de máquina en standby
      ALIMENTAR : Bool;   // Actuador que engloba la operacion de alimentar del brazo (por la cinta superior)
      EXTRAER_POR_ARRIBA : Bool;   // Actuador que engloba la operacion de extracción de piezas del brazo
      EXTRAER_POR_DEBAJO : Bool;   // Actuador que engloba la operacion de extracción de piezas del brazo
   END_VAR
   VAR_IN_OUT
      aviso_defecto : Bool;   // Aviso de defecto (de utilidad para el rearme)
   END_VAR
   VAR
      X_standby : Bool;   // Estado de espera
      X_alimentar : Bool;   // Estado de trabajo
      X_descarga_superior : Bool;   // Estado de trabajo
      X_descarga_inferior : Bool;   // Estado de trabajo
      X_defecto_tiempo : Bool;   // Estado de defecto por tiempo sobrepasado
      X_defecto_emergencia : Bool;   // Estado de defecto por emergencia
      X_defecto_posición : Bool;   // Estado de defecto por mal posicionamiento
      bit_de_trabajo : Bool;   // Bit de trabajo para el arranque
      M_flanco_rearme : Bool;   // Marca de flanco de la señal de rearme
      M_flanco_defecto : Bool;   // Marca de flanco del aviso de defecto
      temporizador : TON_TIME;   // TON para el defecto de tiempo
      M_flanco_orden_alimentar : Bool;   // Marca de flanco para la señal de inicio de la maniobra de alimentación
      M_flanco_fin_maniobra : Bool;   // Marca de flanco de la señal fin_maniobra
   END_VAR
   VAR_TEMP
      aviso_trabajo : Bool;   // Aviso de que la máquina está trabajando (para el disparo del temporizador)
      M_pulso_fin_maniobra : Bool;   // Marca de pulso de la señal fin_maniobra
   END_VAR
   VAR_TEMP   // added for the SCL form of the ladder/FBD networks
      _w1 : Bool;
   END_VAR
BEGIN

REGION Network 1 (STL): DESCONEXIÓN (Start:=False)
   // Aagado de la máquina, máxima prioridad. Se llama a las maniobras con RESET:=TRUE (en caso de haberlas).
   // Tan solo se ponen a cero las salidas, los estados internos se inicializarán en el arranque.
         AN    #Start;
         R     #bit_de_trabajo;
         R     #aviso_standby;
         R     #ALIMENTAR;
         R     #EXTRAER_POR_ARRIBA;
         R     #EXTRAER_POR_DEBAJO;
         R     #aviso_defecto;
         BEC;
END_REGION

REGION Network 2 (STL): DEFECTO (emergencia)
   // Defecto prioritario. LLamamos a las maniobras con RESET:=TRUE (en caso de haberlas)
         A     #EMER;
         S     #X_defecto_emergencia;
         R     #X_standby;
         R     #X_defecto_tiempo;
         R     #X_defecto_posición;
         R     #X_alimentar;
         R     #X_descarga_inferior;
         R     #X_descarga_superior;
END_REGION

REGION Network 3 (STL): DEFECTO (tiempo excedido)
   // Ante el aviso de defecto por tiempo se accede al estado de defecto.
         A     #temporizador.Q;
         S     #X_defecto_tiempo;
         R     #X_alimentar;
         R     #X_descarga_inferior;
         R     #X_descarga_superior;
END_REGION

REGION Network 4 (STL): DEFECTO (mal posicionamiento en el arranque)
   // Si al arrancar, la máquina no está posicionada correctamente, se accede al correspondiente estado de defecto.
         A     #X_standby;
         AN    #brazo_en_posición;
         S     #X_defecto_posición;
         R     #X_standby;
END_REGION

REGION Network 5 (STL): Aviso de defecto (para el rearme)
   // Se avisará al usuario cuando la máquina haya entrado en defecto. El aviso será de utilidad para el rearme.
         A     #X_defecto_posición;
         O     #X_defecto_tiempo;
         FP    #M_flanco_defecto;
         S     #aviso_defecto;
END_REGION

REGION Network 6 (STL): REARME (emergencia)
   // Una vez se ha solucionado el problema  se vuelve al reposo con el flanco positivo de la señal rearme.
         A     #Rearme;
         FP    #M_flanco_rearme;
         A     #X_defecto_emergencia;
         AN    #EMER;
         S     #X_standby;
         R     #X_defecto_emergencia;
END_REGION

REGION Network 7: REARME (Defecto de tiempo o posición)
   // Una vez se ha solucionado el problema, se vuelve al reposo al desactivarse el aviso de error (por el usuario)
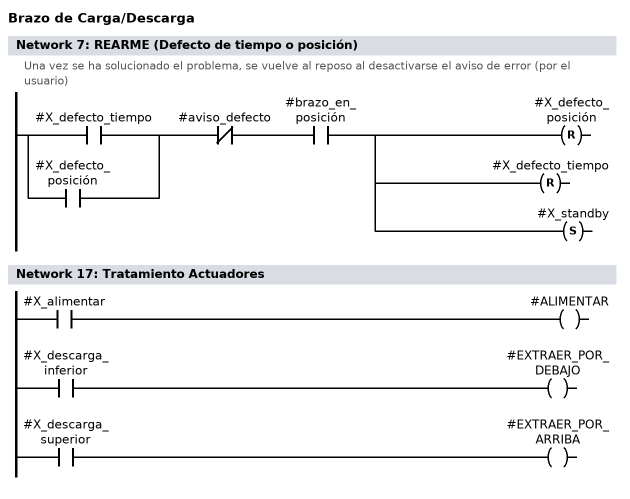
   RUNG wire#powerrail
      Contact( #X_defecto_tiempo )
      wire#w1
      I_Contact( #aviso_defecto )
      Contact( #brazo_en_posición )
      wire#w2
      R_Coil( #X_defecto_posición )
   END_RUNG
   RUNG wire#powerrail
      Contact( #X_defecto_posición )
   END_RUNG wire#w1
   RUNG wire#w2
      R_Coil( #X_defecto_tiempo )
   END_RUNG
   RUNG wire#w2
      S_Coil( #X_standby )
   END_RUNG
   // the same network as SCL:
   #_w1 := (#X_defecto_tiempo OR #X_defecto_posición) AND NOT #aviso_defecto AND #brazo_en_posición;
   IF #_w1 THEN
       #X_defecto_posición := FALSE;
       #X_defecto_tiempo := FALSE;
       #X_standby := TRUE;
   END_IF;
END_REGION

REGION Network 8 (STL): ARRANQUE
   // Arrancamos la máquina, inicializando el estado de standby (X0)
         A     #Start;
         FP    #bit_de_trabajo;
         S     #X_standby;
         R     #X_alimentar;
         R     #X_descarga_inferior;
         R     #X_descarga_superior;
         R     #X_defecto_tiempo;
         R     #X_defecto_emergencia;
         R     #X_defecto_posición;
         R     #M_flanco_defecto;
         R     #M_flanco_rearme;
         R     #aviso_trabajo;
END_REGION

REGION Network 9 (STL): Configuración del Aviso de trabajo para el disparo del temporizador
   // Se usará dicha señal para el disparo del temporizador
         A     #X_alimentar;
         O     #X_descarga_inferior;
         O     #X_descarga_superior;
         =     #aviso_trabajo;
END_REGION

REGION Network 10 (STL): Configuración Temporizador (tiempo límite)
   // Se empleará un TON (sin memoria). Se dispara por cualquiera de los bits de estado de trabajo, asumiendo que las tres maniobras tienen el mismo límite de tiempo.
         CALL  #temporizador
         ( IN := #aviso_trabajo,
           PT := #tiempo,
           Q  := ,
           ET :=
         );
END_REGION

REGION Network 11 (STL): X_Standby -> X_Alimentar
   // El brazo comienza la maniobra de alimentación cuando recibe la orden (orden_alimentar:=TRUE). Se comprobará que el brazo esté correctamente posicionado y que el modo de marcha permita la alimentación (flag_alim:=TRUE)
         A     #orden_alimentar;
         FP    #M_flanco_orden_alimentar;
         A     #X_standby;
         A     #flag_alim;
         A     #brazo_en_posición;
         R     #X_standby;
         S     #X_alimentar;
END_REGION

REGION Network 12 (STL): X_Standby -> X_Descarga_Superior
   // El brazo comienza la maniobra de extracción cuando detecta que ha llegado una pieza (S_superior==TRUE). Se comprobará que el brazo esté correctamente posicionado y que el modo de marcha permita la extracción por la cinta correspondiente (flag_extr_sup==TRUE).
         A     #X_standby;
         A     #S_superior;
         A     #flag_extr_sup;
         A     #brazo_en_posición;
         R     #X_standby;
         S     #X_descarga_superior;
END_REGION

REGION Network 13 (STL): X_Standby -> X_Descarga_Inferior
   // El brazo comienza la maniobra de extracción cuando detecta que ha llegado una pieza (S_inferior==TRUE). Se comprobará que el brazo esté correctamente posicionado y que el modo de marcha permita la extracción por la cinta correspondiente (flag_extr_inf==TRUE).
         A     #X_standby;
         A     #S_inferior;
         A     #flag_extr_inf;
         A     #brazo_en_posición;
         R     #X_standby;
         S     #X_descarga_inferior;
END_REGION

REGION Network 14 (STL): Gestión Flanco Señal fin_maniobra
         A     #fin_maniobra;
         FP    #M_flanco_fin_maniobra;
         =     #M_pulso_fin_maniobra;
END_REGION

REGION Network 15 (STL): Vuelta al reposo
   // Vuelta al reposo al completar cualquiera de las maniobras.
         A     #X_descarga_inferior;
         O     #X_descarga_superior;
         O     #X_alimentar;
         A     #M_pulso_fin_maniobra;
         A     #brazo_en_posición;
         R     #X_alimentar;
         R     #X_descarga_inferior;
         R     #X_descarga_superior;
         S     #X_standby;
END_REGION

REGION Network 16 (STL): Aviso de Standby (para el usuario)
   // Avisa de que la máquina está en standby y funcionando correctamente
         A     #X_standby;
         =     #aviso_standby;
END_REGION

REGION Network 17: Tratamiento Actuadores
   RUNG wire#powerrail
      Contact( #X_alimentar )
      Coil( #ALIMENTAR )
   END_RUNG
   RUNG wire#powerrail
      Contact( #X_descarga_inferior )
      Coil( #EXTRAER_POR_DEBAJO )
   END_RUNG
   RUNG wire#powerrail
      Contact( #X_descarga_superior )
      Coil( #EXTRAER_POR_ARRIBA )
   END_RUNG
   // the same network as SCL:
   #ALIMENTAR := #X_alimentar;
   #EXTRAER_POR_DEBAJO := #X_descarga_inferior;
   #EXTRAER_POR_ARRIBA := #X_descarga_superior;
END_REGION
END_FUNCTION_BLOCK

FUNCTION_BLOCK "Cinta de Volcado (Aviso de Disponibilidad)"   // FB7, LAD
TITLE = Control de la ocupación de la cinta de evacuación de piezas.
{ S7_Optimized_Access := 'TRUE' }
VERSION : 0.1
// Al terminar una máquina de tratar una pieza, ésta deberá ser evacuada. La cinta de volcado propia de cada máquina deberá incorporar la pieza a la cinta de evacuación (que recibe las piezas de todas las máquinas) sin que colisione con piezas ya presentes en la cinta.
// Este bloque se ocupa de gestionar el aviso que indicará que la cinta de evacuación está despejada y es seguro incoporar una pieza.
// NOTA: Este bloque no acaba de seguir el prototipo de "maniobra", ya que no maneja actuadores. Aún así, se ha seguido más o menos la plantilla de "maniobra" dada en las clases de teroría.
// (BLOQUE AUTOCONTENIDO)
   VAR_INPUT
      S_izquierda : Bool;   // Sensor de presencia dela cinta a la que se quiere incorporar la pieza (a la izquierda de la intersección)
      S_derecha : Bool;   // Sensor de presencia dela cinta a la que se quiere incorporar la pieza (a la derecha de la intersección)
      tiempo_limite : Time;   // tiempo límite antes de considerar que la intersección está despejada
      RESET : Bool;   // entrada asíncrona, parada brusca de maniobra
      flag_sentido_cinta_inferior : Bool;   // Vale 1 cuando la cinta se mueve de izquierda a derecha (definido según el modo de marcha)
   END_VAR
   VAR_OUTPUT
      aviso_intersección_libre : Bool;   // Aviso de que es seguro incorporar una pieza
   END_VAR
   VAR
      X3 : Bool;   // Estado de espera (no es seguro incorporar una pieza)
      X4 : Bool;   // Estado de seguridad (ha pasado el tiempo especificado desde la última detección)
      X5 : Bool;   // Estado de paso. Se ha detectado una pieza, se abandonará el estado cuando el sensor deje de detectar la pieza.
      bit_de_trabajo : Bool;   // plantilla arranque
      temporizador : TON_TIME;   // TON para la cuenta
   END_VAR
   VAR_TEMP
      aviso_pieza_detectada : Bool;   // Según el setido de las cintas, almacena la señal del sensor de presencia correspondiente.
   END_VAR
BEGIN

REGION Network 1 (STL): DESCONEXION RESET (prioridad máxima)
   // Desconexión prioritaria.
         A     #RESET;
         JCN   _007;
         CALL  RESET_TIMER
         ( "TIMER" := #temporizador
         );
         A     #RESET;
         R     #bit_de_trabajo;
         R     #aviso_intersección_libre;
         BEC;
   _007: NOP   0;
END_REGION

REGION Network 2 (STL): CONEXIÓN: activación de X_MAN (maniobra simple)
   // Inicialización de los estados.
         SET;
         FP    #bit_de_trabajo;
         S     #X3;
         R     #X4;
         R     #X5;
END_REGION

REGION Network 3: Gestión de la señal de aviso de pieza detectada
   // La señal de aviso dependerá del sentido de las cintas (sentido en el que se aproximan las piezas). Si las piezas provienen de la izquierda, la señal se activará cuando el sensor izquierdo detecte presencia.
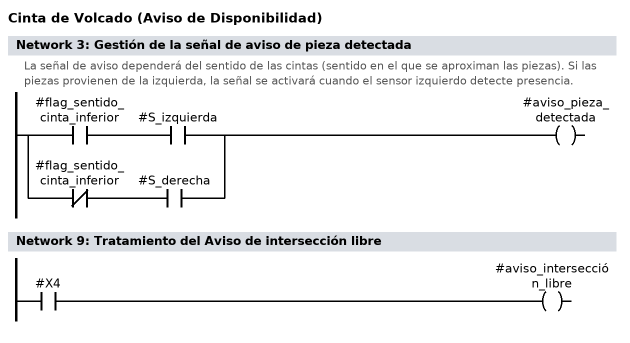
   RUNG wire#powerrail
      Contact( #flag_sentido_cinta_inferior )
      Contact( #S_izquierda )
      wire#w1
      Coil( #aviso_pieza_detectada )
   END_RUNG
   RUNG wire#powerrail
      I_Contact( #flag_sentido_cinta_inferior )
      Contact( #S_derecha )
   END_RUNG wire#w1
   // the same network as SCL:
   #aviso_pieza_detectada := (#flag_sentido_cinta_inferior AND #S_izquierda) OR (NOT #flag_sentido_cinta_inferior AND #S_derecha);
END_REGION

REGION Network 4 (STL): X3->X4
   // Cuando transcurre el tiempo de seguridad, se accede al estado X2, que indica que es seguro incorporar piezas a la cinta de evacuación.
         A     #X3;
         A     #temporizador.Q;
         AN    #aviso_pieza_detectada;
         R     #X3;
         S     #X4;
END_REGION

REGION Network 5 (STL): X3->X5
   // Si antes de que concluyael tiempo de espera se detecta una nueva pieza, se accede a un estado de paso antes de reiniciar la cuenta.
         A     #X3;
         A     #aviso_pieza_detectada;
         R     #X3;
         S     #X5;
END_REGION

REGION Network 6 (STL): X4->X5
   // Si se vuelve a detectar una pieza, se accede al estado de paso antes de reiniciar la cuenta.
         A     #X4;
         A     #aviso_pieza_detectada;
         R     #X4;
         S     #X5;
END_REGION

REGION Network 7 (STL): X5->X3
   // Cuando el aviso desaparezce (la pieza sobrepasa el sensor) se vuelve al estado de espera para reiniciar la cuenta.
         A     #X5;
         AN    #aviso_pieza_detectada;
         R     #X5;
         S     #X3;
END_REGION

REGION Network 8 (STL): CONFIGURACIÓN TEMPORIZADOR
   // Emplearemos un temporizador IEC TON.
         CALL  #temporizador
         ( IN := #X3,
           PT := #tiempo_limite,
           Q  := ,
           ET :=
         );
END_REGION

REGION Network 9: Tratamiento del Aviso de intersección libre
   RUNG wire#powerrail
      Contact( #X4 )
      Coil( #aviso_intersección_libre )
   END_RUNG
   // the same network as SCL:
   #aviso_intersección_libre := #X4;
END_REGION
END_FUNCTION_BLOCK

